C03659=1179.492,110.522,-52.209,-178.814,6.218,148.772
C03660=1179.488,110.772,-52.228,-178.811,6.218,148.772
C03661=1179.483,111.021,-52.246,-178.809,6.220,148.771
C03662=1179.478,111.270,-52.266,-178.806,6.222,148.771
C03663=1179.473,111.519,-52.285,-178.803,6.222,148.770
C03664=1179.468,111.769,-52.304,-178.801,6.224,148.770
C03665=1179.463,112.018,-52.323,-178.799,6.225,148.769
C03666=1179.459,112.267,-52.342,-178.795,6.226,148.769
C03667=1179.453,112.517,-52.361,-178.793,6.228,148.768
C03668=1179.449,112.765,-52.379,-178.790,6.229,148.768
C03669=1179.444,113.015,-52.399,-178.787,6.230,148.767
C03670=1179.439,113.263,-52.418,-178.785,6.232,148.767
C03671=1179.434,113.514,-52.437,-178.782,6.233,148.767
C03672=1179.429,113.762,-52.456,-178.779,6.234,148.766
C03673=1179.425,114.012,-52.475,-178.777,6.236,148.765
C03674=1179.420,114.260,-52.494,-178.774,6.237,148.765
C03675=1179.415,114.510,-52.514,-178.771,6.239,148.764
C03676=1179.410,114.759,-52.532,-178.769,6.240,148.764
C03677=1179.405,115.009,-52.552,-178.766,6.241,148.764
C03678=1179.401,115.257,-52.570,-178.764,6.243,148.763
C03679=1179.396,115.507,-52.590,-178.761,6.244,148.763
C03680=1179.390,115.756,-52.609,-178.758,6.245,148.762
C03681=1179.386,116.005,-52.628,-178.756,6.247,148.762
C03682=1179.382,116.255,-52.648,-178.752,6.248,148.761
C03683=1179.376,116.504,-52.666,-178.750,6.249,148.761
C03684=1179.372,116.753,-52.686,-178.748,6.251,148.760
C03685=1179.367,117.002,-52.705,-178.744,6.252,148.760
C03686=1179.362,117.252,-52.724,-178.742,6.253,148.759
C03687=1179.357,117.501,-52.744,-178.740,6.255,148.759
C03688=1179.353,117.750,-52.763,-178.737,6.257,148.759
C03689=1179.347,117.999,-52.782,-178.734,6.257,148.758
C03690=1179.343,118.248,-52.802,-178.732,6.259,148.757
C03691=1179.339,118.498,-52.821,-178.729,6.261,148.757
C03692=1179.333,118.746,-52.840,-178.726,6.261,148.756
C03693=1179.328,118.996,-52.860,-178.724,6.263,148.756
C03694=1179.323,119.245,-52.879,-178.721,6.265,148.756
C03695=1179.319,119.494,-52.898,-178.718,6.267,148.755
C03696=1179.314,119.744,-52.918,-178.716,6.267,148.755
C03697=1179.309,119.993,-52.937,-178.713,6.269,148.754
C03698=1179.304,120.242,-52.957,-178.710,6.271,148.754
C03699=1179.299,120.491,-52.976,-178.708,6.271,148.753
C03700=1179.295,120.740,-52.995,-178.705,6.273,148.753
C03701=1179.290,120.990,-53.015,-178.702,6.275,148.752
C03702=1179.285,121.239,-53.034,-178.700,6.276,148.752
C03703=1179.280,121.488,-53.054,-178.697,6.277,148.751
C03704=1179.276,121.737,-53.074,-178.694,6.279,148.751
C03705=1179.271,121.986,-53.093,-178.691,6.280,148.751
C03706=1179.266,122.235,-53.112,-178.689,6.281,148.750
C03707=1179.261,122.484,-53.132,-178.686,6.283,148.750
C03708=1179.256,122.734,-53.151,-178.683,6.284,148.749
C03709=1179.251,122.983,-53.171,-178.681,6.285,148.749
C03710=1179.246,123.232,-53.190,-178.679,6.287,148.748
C03711=1179.242,123.481,-53.211,-178.675,6.289,148.748
C03712=1179.238,123.730,-53.230,-178.673,6.290,148.747
C03713=1179.232,123.979,-53.249,-178.671,6.291,148.747
C03714=1179.228,124.229,-53.269,-178.667,6.293,148.746
C03715=1179.223,124.478,-53.288,-178.665,6.294,148.746
C03716=1179.218,124.727,-53.309,-178.663,6.295,148.745
C03717=1179.213,124.976,-53.328,-178.660,6.297,148.745
C03718=1179.208,125.226,-53.348,-178.657,6.298,148.744
C03719=1179.204,125.475,-53.367,-178.654,6.300,148.744
C03720=1179.199,125.724,-53.387,-178.652,6.301,148.744
C03721=1179.194,125.973,-53.407,-178.649,6.303,148.743
C03722=1179.189,126.223,-53.427,-178.646,6.304,148.743
C03723=1179.185,126.472,-53.447,-178.643,6.306,148.742
C03724=1179.179,126.721,-53.466,-178.641,6.307,148.742
C03725=1179.175,126.970,-53.485,-178.638,6.309,148.741
C03726=1179.171,127.219,-53.506,-178.636,6.310,148.741
C03727=1179.165,127.468,-53.525,-178.633,6.312,148.740
C03728=1179.161,127.717,-53.545,-178.630,6.313,148.740
C03729=1179.156,127.966,-53.565,-178.628,6.314,148.740
C03730=1179.152,128.216,-53.585,-178.625,6.316,148.739
C03731=1179.147,128.465,-53.604,-178.622,6.318,148.739
C03732=1179.142,128.714,-53.624,-178.620,6.318,148.738
C03733=1179.137,128.963,-53.644,-178.617,6.320,148.738
C03734=1179.133,129.212,-53.664,-178.614,6.322,148.737
C03735=1179.127,129.462,-53.685,-178.611,6.323,148.737
C03736=1179.122,129.711,-53.704,-178.609,6.324,148.736
C03737=1179.117,129.960,-53.724,-178.606,6.326,148.736
C03738=1179.113,130.209,-53.744,-178.604,6.328,148.736
C03739=1179.108,130.458,-53.764,-178.601,6.329,148.735
C03740=1179.103,130.708,-53.784,-178.598,6.331,148.735
C03741=1179.098,130.956,-53.804,-178.596,6.332,148.734
C03742=1179.094,131.206,-53.824,-178.593,6.334,148.734
C03743=1179.089,131.455,-53.844,-178.590,6.335,148.733
C03744=1179.084,131.704,-53.864,-178.587,6.337,148.733
C03745=1179.080,131.953,-53.884,-178.585,6.338,148.732
C03746=1179.074,132.222,-53.906,-178.582,6.339,148.732
C03747=1179.070,132.490,-53.928,-178.579,6.341,148.732
C03748=1179.064,132.759,-53.949,-178.576,6.343,148.731
C03749=1179.059,133.028,-53.970,-178.574,6.344,148.731
C03750=1179.054,133.277,-53.991,-178.571,6.346,148.730
C03751=1179.049,133.525,-54.011,-178.568,6.347,148.730
C03752=1179.044,133.775,-54.031,-178.565,6.349,148.729
C03753=1179.040,134.024,-54.051,-178.562,6.351,148.729
C03754=1179.035,134.273,-54.071,-178.560,6.352,148.728
C03755=1179.031,134.522,-54.091,-178.558,6.354,148.728
C03756=1179.025,134.772,-54.112,-178.554,6.355,148.727
C03757=1179.021,135.021,-54.132,-178.552,6.357,148.727
C03758=1179.016,135.269,-54.152,-178.549,6.358,148.727
C03759=1179.011,135.518,-54.172,-178.547,6.359,148.726
C03760=1179.006,135.768,-54.192,-178.544,6.361,148.726
C03761=1179.001,136.017,-54.213,-178.541,6.363,148.725
C03762=1178.997,136.266,-54.233,-178.538,6.364,148.725
C03763=1178.992,136.515,-54.254,-178.536,6.366,148.724
C03764=1178.988,136.765,-54.273,-178.533,6.367,148.724
C03765=1178.983,137.014,-54.294,-178.531,6.369,148.724
C03766=1178.978,137.263,-54.315,-178.528,6.370,148.723
C03767=1178.974,137.512,-54.335,-178.525,6.372,148.723
C03768=1178.968,137.762,-54.355,-178.522,6.374,148.722
C03769=1178.964,138.011,-54.376,-178.520,6.375,148.722
C03770=1178.959,138.259,-54.396,-178.517,6.376,148.721
C03771=1178.954,138.508,-54.416,-178.515,6.378,148.721
C03772=1178.949,138.757,-54.437,-178.512,6.380,148.721
C03773=1178.944,139.007,-54.457,-178.509,6.381,148.720
C03774=1178.940,139.256,-54.477,-178.506,6.383,148.720
C03775=1178.935,139.505,-54.498,-178.504,6.384,148.719
C03776=1178.930,139.754,-54.518,-178.501,6.386,148.719
C03777=1178.926,140.003,-54.539,-178.499,6.387,148.719
C03778=1178.921,140.252,-54.560,-178.496,6.389,148.718
C03779=1178.916,140.501,-54.580,-178.493,6.391,148.718
C03780=1178.912,140.750,-54.601,-178.490,6.392,148.717
C03781=1178.906,141.000,-54.621,-178.488,6.393,148.717
C03782=1178.902,141.249,-54.641,-178.485,6.395,148.716
C03783=1178.897,141.498,-54.662,-178.482,6.397,148.716
C03784=1178.892,141.747,-54.682,-178.480,6.398,148.716
C03785=1178.888,141.996,-54.703,-178.477,6.400,148.715
C03786=1178.883,142.245,-54.724,-178.474,6.402,148.715
C03787=1178.878,142.494,-54.744,-178.472,6.403,148.714
C03788=1178.873,142.743,-54.765,-178.469,6.404,148.714
C03789=1178.869,142.992,-54.786,-178.466,6.406,148.713
C03790=1178.864,143.241,-54.806,-178.464,6.408,148.713
C03791=1178.859,143.491,-54.827,-178.461,6.410,148.713
C03792=1178.855,143.739,-54.847,-178.458,6.411,148.712
C03793=1178.849,143.989,-54.868,-178.456,6.413,148.712
C03794=1178.845,144.238,-54.889,-178.453,6.414,148.711
C03795=1178.840,144.488,-54.910,-178.450,6.415,148.711
C03796=1178.836,144.736,-54.931,-178.448,6.417,148.711
C03797=1178.831,144.985,-54.952,-178.445,6.419,148.710
C03798=1178.827,145.234,-54.972,-178.442,6.421,148.710
C03799=1178.821,145.483,-54.993,-178.440,6.422,148.709
C03800=1178.817,145.732,-55.014,-178.437,6.424,148.709
C03801=1178.812,145.982,-55.035,-178.434,6.426,148.709
C03802=1178.807,146.231,-55.055,-178.432,6.427,148.708
C03803=1178.802,146.480,-55.076,-178.429,6.428,148.708
C03804=1178.798,146.728,-55.097,-178.426,6.430,148.707
C03805=1178.793,146.977,-55.118,-178.424,6.432,148.707
C03806=1178.788,147.226,-55.138,-178.421,6.434,148.706
C03807=1178.784,147.476,-55.160,-178.418,6.435,148.706
C03808=1178.779,147.726,-55.181,-178.415,6.437,148.706
C03809=1178.774,147.975,-55.201,-178.413,6.439,148.705
C03810=1178.769,148.223,-55.223,-178.410,6.441,148.705
C03811=1178.765,148.472,-55.243,-178.407,6.441,148.704
C03812=1178.760,148.721,-55.264,-178.405,6.443,148.704
C03813=1178.755,148.971,-55.285,-178.402,6.445,148.704
C03814=1178.751,149.219,-55.306,-178.399,6.446,148.703
C03815=1178.746,149.469,-55.327,-178.397,6.448,148.703
C03816=1178.742,149.718,-55.348,-178.394,6.450,148.702
C03817=1178.737,149.967,-55.370,-178.391,6.452,148.702
C03818=1178.731,150.216,-55.390,-178.389,6.453,148.702
C03819=1178.727,150.465,-55.411,-178.386,6.455,148.701
C03820=1178.722,150.713,-55.433,-178.383,6.457,148.701
C03821=1178.718,150.963,-55.454,-178.381,6.458,148.700
C03822=1178.713,151.212,-55.474,-178.378,6.459,148.700
C03823=1178.708,151.461,-55.496,-178.375,6.461,148.700
C03824=1178.703,151.710,-55.517,-178.373,6.463,148.699
C03825=1178.699,151.959,-55.537,-178.370,6.465,148.699
C03826=1178.694,152.209,-55.559,-178.367,6.466,148.698
C03827=1178.689,152.458,-55.580,-178.365,6.468,148.698
C03828=1178.684,152.706,-55.602,-178.362,6.470,148.698
C03829=1178.680,152.955,-55.622,-178.359,6.472,148.697
C03830=1178.675,153.204,-55.644,-178.356,6.473,148.697
C03831=1178.670,153.454,-55.665,-178.354,6.475,148.696
C03832=1178.665,153.703,-55.686,-178.351,6.477,148.696
C03833=1178.661,153.952,-55.707,-178.349,6.478,148.696
C03834=1178.656,154.201,-55.728,-178.346,6.480,148.695
C03835=1178.652,154.450,-55.750,-178.343,6.481,148.695
C03836=1178.647,154.699,-55.771,-178.340,6.483,148.694
C03837=1178.642,154.948,-55.792,-178.338,6.485,148.694
C03838=1178.637,155.197,-55.813,-178.335,6.486,148.694
C03839=1178.633,155.446,-55.835,-178.332,6.488,148.693
C03840=1178.628,155.695,-55.857,-178.330,6.490,148.693
C03841=1178.623,155.944,-55.878,-178.327,6.492,148.692
C03842=1178.618,156.193,-55.900,-178.324,6.493,148.692
C03843=1178.614,156.443,-55.921,-178.322,6.495,148.692
C03844=1178.609,156.691,-55.942,-178.319,6.497,148.691
C03845=1178.604,156.940,-55.963,-178.316,6.499,148.691
C03846=1178.599,157.189,-55.985,-178.314,6.500,148.691
C03847=1178.595,157.438,-56.007,-178.311,6.502,148.690
C03848=1178.590,157.688,-56.028,-178.308,6.504,148.690
C03849=1178.586,157.936,-56.049,-178.305,6.506,148.689
C03850=1178.580,158.205,-56.072,-178.303,6.507,148.689
C03851=1178.576,158.474,-56.096,-178.300,6.509,148.689
C03852=1178.570,158.743,-56.119,-178.297,6.511,148.688
C03853=1178.566,159.012,-56.142,-178.294,6.512,148.688
C03854=1178.561,159.261,-56.164,-178.292,6.514,148.687
C03855=1178.556,159.510,-56.186,-178.289,6.516,148.687
C03856=1178.551,159.759,-56.207,-178.286,6.518,148.687
C03857=1178.546,160.008,-56.228,-178.284,6.519,148.686
C03858=1178.542,160.257,-56.250,-178.281,6.521,148.686
C03859=1178.537,160.506,-56.272,-178.278,6.523,148.686
C03860=1178.533,160.756,-56.293,-178.275,6.525,148.685
C03861=1178.528,161.005,-56.315,-178.273,6.527,148.685
C03862=1178.523,161.253,-56.337,-178.270,6.528,148.684
C03863=1178.519,161.503,-56.359,-178.267,6.530,148.684
C03864=1178.514,161.751,-56.380,-178.265,6.532,148.684
C03865=1178.509,162.001,-56.401,-178.262,6.534,148.683
C03866=1178.504,162.250,-56.424,-178.259,6.535,148.683
C03867=1178.499,162.499,-56.445,-178.257,6.537,148.683
C03868=1178.495,162.748,-56.467,-178.254,6.539,148.682
C03869=1178.490,162.997,-56.489,-178.251,6.541,148.682
C03870=1178.485,163.245,-56.511,-178.249,6.542,148.681
C03871=1178.481,163.494,-56.533,-178.246,6.544,148.681
C03872=1178.476,163.744,-56.554,-178.243,6.546,148.681
C03873=1178.472,163.993,-56.576,-178.241,6.548,148.680
C03874=1178.467,164.242,-56.597,-178.238,6.549,148.680
C03875=1178.463,164.491,-56.619,-178.235,6.551,148.680
C03876=1178.458,164.740,-56.641,-178.233,6.553,148.679
C03877=1178.453,164.988,-56.663,-178.230,6.555,148.679
C03878=1178.449,165.238,-56.685,-178.227,6.557,148.678
C03879=1178.443,165.487,-56.707,-178.224,6.558,148.678
C03880=1178.439,165.736,-56.729,-178.222,6.560,148.678
C03881=1178.434,165.985,-56.751,-178.219,6.562,148.677
C03882=1178.430,166.234,-56.773,-178.216,6.564,148.677
C03883=1178.425,166.483,-56.795,-178.214,6.565,148.677
C03884=1178.420,166.732,-56.817,-178.211,6.567,148.676
C03885=1178.416,166.981,-56.838,-178.208,6.569,148.676
C03886=1178.411,167.230,-56.860,-178.206,6.571,148.676
C03887=1178.406,167.479,-56.883,-178.203,6.572,148.675
C03888=1178.402,167.728,-56.905,-178.200,6.574,148.675
C03889=1178.397,167.976,-56.927,-178.198,6.576,148.674
C03890=1178.393,168.226,-56.949,-178.195,6.578,148.674
C03891=1178.388,168.474,-56.971,-178.192,6.580,148.674
C03892=1178.383,168.724,-56.993,-178.190,6.581,148.673
C03893=1178.378,168.973,-57.015,-178.187,6.583,148.673
C03894=1178.374,169.222,-57.037,-178.184,6.585,148.673
C03895=1178.369,169.470,-57.059,-178.182,6.587,148.672
C03896=1178.365,169.719,-57.082,-178.179,6.588,148.672
C03897=1178.359,169.968,-57.104,-178.176,6.591,148.672
C03898=1178.355,170.218,-57.126,-178.173,6.593,148.671
C03899=1178.350,170.466,-57.148,-178.170,6.595,148.671
C03900=1178.346,170.715,-57.170,-178.168,6.596,148.670
C03901=1178.340,170.964,-57.193,-178.165,6.598,148.670
C03902=1178.336,171.213,-57.215,-178.163,6.600,148.670
C03903=1178.331,171.462,-57.236,-178.160,6.602,148.670
C03904=1178.326,171.711,-57.259,-178.157,6.604,148.669
C03905=1178.322,171.960,-57.282,-178.155,6.606,148.669
C03906=1178.318,172.209,-57.303,-178.152,6.607,148.668
C03907=1178.313,172.458,-57.326,-178.149,6.609,148.668
C03908=1178.308,172.706,-57.349,-178.147,6.611,148.668
C03909=1178.304,172.956,-57.371,-178.144,6.613,148.667
C03910=1178.299,173.205,-57.393,-178.141,6.614,148.667
C03911=1178.294,173.453,-57.416,-178.139,6.616,148.667
C03912=1178.290,173.703,-57.438,-178.136,6.618,148.666
C03913=1178.285,173.951,-57.459,-178.133,6.620,148.666
C03914=1178.280,174.201,-57.483,-178.131,6.621,148.666
C03915=1178.276,174.450,-57.505,-178.127,6.624,148.665
C03916=1178.270,174.699,-57.527,-178.125,6.626,148.665
C03917=1178.266,174.948,-57.550,-178.122,6.628,148.665
C03918=1178.262,175.197,-57.572,-178.120,6.630,148.664
C03919=1178.257,175.445,-57.595,-178.117,6.631,148.664
C03920=1178.253,175.695,-57.617,-178.114,6.633,148.664
C03921=1178.247,175.943,-57.640,-178.112,6.635,148.663
C03922=1178.243,176.192,-57.662,-178.109,6.637,148.663
C03923=1178.239,176.442,-57.684,-178.106,6.639,148.663
C03924=1178.233,176.690,-57.707,-178.104,6.640,148.662
C03925=1178.229,176.939,-57.729,-178.101,6.642,148.662
C03926=1178.224,177.188,-57.752,-178.098,6.644,148.661
C03927=1178.220,177.436,-57.775,-178.095,6.647,148.661
C03928=1178.215,177.686,-57.797,-178.093,6.649,148.661
C03929=1178.211,177.935,-57.820,-178.090,6.650,148.661
C03930=1178.206,178.184,-57.843,-178.087,6.652,148.660
C03931=1178.201,178.432,-57.865,-178.085,6.654,148.660
C03932=1178.196,178.682,-57.888,-178.082,6.656,148.659
C03933=1178.192,178.931,-57.911,-178.079,6.658,148.659
C03934=1178.187,179.180,-57.933,-178.077,6.659,148.659
C03935=1178.183,179.428,-57.956,-178.074,6.661,148.658
C03936=1178.178,179.677,-57.979,-178.071,6.663,148.658
C03937=1178.174,179.927,-58.001,-178.069,6.666,148.658
C03938=1178.169,180.175,-58.024,-178.066,6.668,148.658
C03939=1178.165,180.424,-58.047,-178.063,6.669,148.657
C03940=1178.160,180.673,-58.069,-178.061,6.671,148.657
C03941=1178.156,180.922,-58.092,-178.058,6.673,148.656
C03942=1178.150,181.170,-58.115,-178.055,6.675,148.656
C03943=1178.145,181.420,-58.138,-178.053,6.676,148.656
C03944=1178.141,181.669,-58.161,-178.050,6.678,148.655
C03945=1178.137,181.918,-58.184,-178.047,6.681,148.655
C03946=1178.132,182.166,-58.206,-178.044,6.683,148.655
C03947=1178.127,182.416,-58.229,-178.042,6.685,148.655
C03948=1178.122,182.665,-58.252,-178.039,6.686,148.654
C03949=1178.118,182.913,-58.275,-178.036,6.688,148.654
C03950=1178.113,183.162,-58.298,-178.034,6.690,148.654
C03951=1178.109,183.411,-58.320,-178.031,6.692,148.653
C03952=1178.104,183.660,-58.344,-178.029,6.694,148.653
C03953=1178.099,183.909,-58.367,-178.026,6.697,148.653
C03954=1178.095,184.179,-58.391,-178.023,6.698,148.652
C03955=1178.090,184.448,-58.416,-178.020,6.700,148.652
C03956=1178.084,184.718,-58.441,-178.017,6.703,148.652
C03957=1178.080,184.987,-58.467,-178.014,6.704,148.651
C03958=1178.075,185.237,-58.489,-178.012,6.706,148.651
C03959=1178.070,185.486,-58.513,-178.008,6.709,148.651
C03960=1178.066,185.734,-58.535,-178.006,6.711,148.650
C03961=1178.061,185.983,-58.558,-178.003,6.712,148.650
C03962=1178.056,186.232,-58.582,-178.000,6.714,148.650
C03963=1178.052,186.481,-58.605,-177.998,6.716,148.649
C03964=1178.048,186.729,-58.628,-177.996,6.718,148.649
C03965=1178.043,186.978,-58.651,-177.993,6.720,148.649
C03966=1178.038,187.227,-58.675,-177.990,6.722,148.648
C03967=1178.033,187.476,-58.698,-177.987,6.724,148.648
C03968=1178.029,187.725,-58.720,-177.984,6.726,148.648
C03969=1178.024,187.974,-58.744,-177.982,6.728,148.648
C03970=1178.020,188.223,-58.767,-177.979,6.730,148.647
C03971=1178.015,188.472,-58.790,-177.977,6.732,148.647
C03972=1178.010,188.721,-58.814,-177.974,6.734,148.646
C03973=1178.006,188.969,-58.836,-177.971,6.736,148.646
C03974=1178.002,189.218,-58.860,-177.969,6.738,148.646
C03975=1177.997,189.467,-58.883,-177.966,6.740,148.646
C03976=1177.992,189.716,-58.907,-177.963,6.742,148.645
C03977=1177.987,189.965,-58.930,-177.960,6.744,148.645
C03978=1177.982,190.214,-58.953,-177.957,6.746,148.645
C03979=1177.978,190.463,-58.976,-177.955,6.748,148.644
C03980=1177.974,190.711,-59.000,-177.953,6.750,148.644
C03981=1177.969,190.960,-59.023,-177.950,6.752,148.644
C03982=1177.964,191.209,-59.046,-177.947,6.754,148.643
C03983=1177.960,191.458,-59.070,-177.944,6.756,148.643
C03984=1177.955,191.707,-59.093,-177.942,6.758,148.643
C03985=1177.950,191.956,-59.117,-177.939,6.760,148.643
C03986=1177.946,192.205,-59.141,-177.936,6.762,148.642
C03987=1177.941,192.454,-59.164,-177.934,6.764,148.642
C03988=1177.936,192.703,-59.187,-177.930,6.766,148.642
C03989=1177.932,192.952,-59.211,-177.928,6.768,148.641
C03990=1177.927,193.200,-59.235,-177.926,6.770,148.641
C03991=1177.923,193.449,-59.258,-177.923,6.772,148.641
C03992=1177.919,193.698,-59.281,-177.920,6.774,148.640
C03993=1177.914,193.947,-59.304,-177.917,6.776,148.640
C03994=1177.910,194.195,-59.328,-177.915,6.779,148.640
C03995=1177.905,194.444,-59.352,-177.912,6.780,148.640
C03996=1177.900,194.693,-59.375,-177.910,6.782,148.639
C03997=1177.896,194.942,-59.399,-177.906,6.785,148.639
C03998=1177.891,195.191,-59.422,-177.904,6.787,148.639
C03999=1177.886,195.440,-59.446,-177.901,6.789,148.638
C04000=1177.882,195.688,-59.470,-177.899,6.790,148.638
C04001=1177.877,195.937,-59.493,-177.896,6.792,148.638
C04002=1177.873,196.186,-59.517,-177.893,6.795,148.638
C04003=1177.868,196.435,-59.541,-177.891,6.797,148.637
C04004=1177.863,196.684,-59.565,-177.888,6.799,148.637
C04005=1177.858,196.932,-59.589,-177.885,6.801,148.637
C04006=1177.854,197.181,-59.612,-177.883,6.803,148.636
C04007=1177.849,197.431,-59.635,-177.880,6.805,148.636
C04008=1177.845,197.679,-59.660,-177.877,6.807,148.636
C04009=1177.840,197.928,-59.683,-177.875,6.809,148.635
C04010=1177.836,198.176,-59.707,-177.872,6.812,148.635
C04011=1177.831,198.426,-59.731,-177.869,6.814,148.635
C04012=1177.827,198.675,-59.755,-177.866,6.815,148.635
C04013=1177.822,198.924,-59.778,-177.864,6.817,148.634
C04014=1177.817,199.172,-59.803,-177.862,6.819,148.634
C04015=1177.813,199.421,-59.826,-177.858,6.822,148.634
C04016=1177.808,199.670,-59.850,-177.856,6.824,148.633
C04017=1177.804,199.918,-59.874,-177.853,6.825,148.633
C04018=1177.799,200.167,-59.898,-177.851,6.828,148.633
C04019=1177.795,200.416,-59.922,-177.848,6.830,148.633
C04020=1177.791,200.665,-59.945,-177.845,6.832,148.632
C04021=1177.785,200.914,-59.970,-177.842,6.834,148.632
C04022=1177.781,201.162,-59.994,-177.839,6.837,148.632
C04023=1177.776,201.411,-60.018,-177.837,6.839,148.632
C04024=1177.772,201.660,-60.042,-177.834,6.840,148.631
C04025=1177.767,201.909,-60.065,-177.832,6.842,148.631
C04026=1177.762,202.158,-60.090,-177.829,6.845,148.631
C04027=1177.758,202.407,-60.114,-177.826,6.847,148.630
C04028=1177.754,202.656,-60.137,-177.823,6.849,148.630
C04029=1177.749,202.904,-60.162,-177.821,6.851,148.630
C04030=1177.744,203.153,-60.186,-177.818,6.853,148.630
C04031=1177.740,203.401,-60.210,-177.815,6.855,148.629
C04032=1177.736,203.651,-60.234,-177.813,6.857,148.629
C04033=1177.731,203.899,-60.258,-177.810,6.859,148.629
C04034=1177.726,204.148,-60.283,-177.807,6.862,148.628
C04035=1177.722,204.397,-60.307,-177.805,6.864,148.628
C04036=1177.717,204.646,-60.330,-177.802,6.866,148.628
C04037=1177.712,204.895,-60.355,-177.799,6.868,148.628
C04038=1177.708,205.143,-60.379,-177.796,6.870,148.627
C04039=1177.704,205.392,-60.403,-177.794,6.872,148.627
C04040=1177.699,205.641,-60.428,-177.792,6.874,148.627
C04041=1177.694,205.889,-60.452,-177.788,6.877,148.627
C04042=1177.690,206.139,-60.476,-177.786,6.879,148.626
C04043=1177.685,206.387,-60.501,-177.784,6.880,148.626
C04044=1177.680,206.636,-60.525,-177.780,6.883,148.626
C04045=1177.676,206.884,-60.549,-177.778,6.885,148.626
C04046=1177.672,207.134,-60.574,-177.775,6.887,148.625
C04047=1177.667,207.382,-60.598,-177.772,6.890,148.625
C04048=1177.662,207.631,-60.622,-177.770,6.892,148.625
C04049=1177.658,207.879,-60.647,-177.767,6.894,148.625
C04050=1177.654,208.128,-60.671,-177.764,6.896,148.624
C04051=1177.649,208.377,-60.696,-177.762,6.898,148.624
C04052=1177.644,208.626,-60.720,-177.759,6.900,148.624
C04053=1177.640,208.875,-60.745,-177.757,6.902,148.623
C04054=1177.635,209.123,-60.769,-177.754,6.905,148.623
C04055=1177.630,209.372,-60.793,-177.751,6.907,148.623
C04056=1177.626,209.620,-60.818,-177.749,6.908,148.623
C04057=1177.621,209.870,-60.843,-177.746,6.911,148.623
C04058=1177.616,210.141,-60.869,-177.743,6.913,148.622
C04059=1177.611,210.411,-60.895,-177.740,6.916,148.622
C04060=1177.607,210.681,-60.922,-177.737,6.918,148.622
C04061=1177.602,210.952,-60.948,-177.734,6.920,148.621
C04062=1177.597,211.200,-60.973,-177.731,6.923,148.621
C04063=1177.593,211.449,-60.998,-177.729,6.925,148.621
C04064=1177.588,211.698,-61.022,-177.726,6.927,148.621
C04065=1177.583,211.947,-61.046,-177.723,6.930,148.620
C04066=1177.579,212.195,-61.072,-177.720,6.931,148.620
C04067=1177.575,212.444,-61.096,-177.718,6.934,148.620
C04068=1177.570,212.693,-61.121,-177.715,6.936,148.620
C04069=1177.565,212.942,-61.146,-177.712,6.938,148.619
C04070=1177.561,213.190,-61.170,-177.710,6.940,148.619
C04071=1177.556,213.440,-61.195,-177.707,6.943,148.619
C04072=1177.552,213.688,-61.220,-177.705,6.945,148.619
C04073=1177.547,213.936,-61.244,-177.702,6.947,148.618
C04074=1177.542,214.186,-61.269,-177.699,6.949,148.618
C04075=1177.538,214.434,-61.294,-177.697,6.951,148.618
C04076=1177.534,214.683,-61.319,-177.694,6.953,148.618
C04077=1177.529,214.931,-61.343,-177.691,6.956,148.617
C04078=1177.524,215.180,-61.368,-177.689,6.958,148.617
C04079=1177.520,215.430,-61.393,-177.686,6.960,148.617
C04080=1177.516,215.677,-61.418,-177.683,6.963,148.617
C04081=1177.511,215.927,-61.443,-177.681,6.965,148.616
C04082=1177.506,216.175,-61.468,-177.677,6.967,148.616
C04083=1177.502,216.424,-61.493,-177.675,6.969,148.616
C04084=1177.497,216.673,-61.517,-177.672,6.971,148.616
C04085=1177.492,216.921,-61.543,-177.670,6.974,148.616
C04086=1177.489,217.170,-61.567,-177.667,6.976,148.615
C04087=1177.484,217.419,-61.592,-177.664,6.978,148.615
C04088=1177.479,217.667,-61.618,-177.662,6.981,148.615
C04089=1177.474,217.916,-61.642,-177.659,6.982,148.615
C04090=1177.471,218.165,-61.667,-177.657,6.985,148.614
C04091=1177.466,218.413,-61.692,-177.654,6.987,148.614
C04092=1177.461,218.663,-61.717,-177.651,6.989,148.614
C04093=1177.456,218.911,-61.743,-177.648,6.992,148.614
C04094=1177.452,219.160,-61.767,-177.645,6.994,148.613
C04095=1177.448,219.408,-61.792,-177.643,6.996,148.613
C04096=1177.443,219.658,-61.817,-177.640,6.998,148.613
C04097=1177.438,219.906,-61.843,-177.638,7.001,148.613
C04098=1177.434,220.155,-61.867,-177.635,7.003,148.613
C04099=1177.430,220.403,-61.893,-177.632,7.005,148.612
C04100=1177.425,220.652,-61.918,-177.630,7.007,148.612
C04101=1177.420,220.900,-61.943,-177.627,7.010,148.612
C04102=1177.416,221.149,-61.969,-177.624,7.012,148.612
C04103=1177.412,221.398,-61.993,-177.621,7.015,148.611
C04104=1177.407,221.646,-62.019,-177.619,7.017,148.611
C04105=1177.403,221.896,-62.044,-177.616,7.019,148.611
C04106=1177.398,222.144,-62.069,-177.613,7.021,148.611
C04107=1177.394,222.393,-62.095,-177.611,7.023,148.610
C04108=1177.389,222.641,-62.119,-177.608,7.026,148.610
C04109=1177.384,222.890,-62.145,-177.606,7.028,148.610
C04110=1177.380,223.138,-62.171,-177.603,7.030,148.610
C04111=1177.376,223.387,-62.195,-177.600,7.033,148.610
C04112=1177.372,223.636,-62.221,-177.597,7.035,148.609
C04113=1177.367,223.884,-62.246,-177.595,7.038,148.609
C04114=1177.362,224.134,-62.271,-177.592,7.039,148.609
C04115=1177.357,224.382,-62.297,-177.589,7.042,148.609
C04116=1177.353,224.631,-62.322,-177.587,7.044,148.609
C04117=1177.349,224.880,-62.348,-177.584,7.046,148.608
C04118=1177.344,225.128,-62.373,-177.581,7.049,148.608
C04119=1177.340,225.377,-62.399,-177.579,7.051,148.608
C04120=1177.335,225.625,-62.424,-177.576,7.054,148.608
C04121=1177.331,225.874,-62.450,-177.574,7.056,148.608
C04122=1177.326,226.123,-62.475,-177.570,7.058,148.607
C04123=1177.321,226.371,-62.500,-177.568,7.060,148.607
C04124=1177.317,226.620,-62.526,-177.566,7.062,148.607
C04125=1177.313,226.869,-62.552,-177.562,7.065,148.607
C04126=1177.308,227.117,-62.577,-177.560,7.067,148.606
C04127=1177.304,227.366,-62.603,-177.557,7.070,148.606
C04128=1177.300,227.615,-62.628,-177.555,7.072,148.606
C04129=1177.295,227.863,-62.654,-177.552,7.074,148.606
C04130=1177.290,228.112,-62.680,-177.549,7.077,148.606
C04131=1177.286,228.361,-62.705,-177.546,7.079,148.605
C04132=1177.281,228.609,-62.730,-177.544,7.081,148.605
C04133=1177.277,228.858,-62.756,-177.542,7.084,148.605
C04134=1177.273,229.107,-62.782,-177.539,7.086,148.605
C04135=1177.268,229.355,-62.807,-177.536,7.088,148.605
C04136=1177.263,229.604,-62.833,-177.533,7.091,148.604
C04137=1177.259,229.853,-62.859,-177.531,7.093,148.604
C04138=1177.254,230.102,-62.885,-177.528,7.096,148.604
C04139=1177.250,230.350,-62.910,-177.526,7.098,148.604
C04140=1177.245,230.599,-62.936,-177.522,7.100,148.604
C04141=1177.241,230.847,-62.962,-177.520,7.103,148.603
C04142=1177.237,231.095,-62.988,-177.517,7.105,148.603
C04143=1177.232,231.344,-63.014,-177.515,7.107,148.603
C04144=1177.227,231.593,-63.040,-177.512,7.110,148.603
C04145=1177.223,231.842,-63.066,-177.509,7.112,148.603
C04146=1177.218,232.090,-63.091,-177.507,7.114,148.602
C04147=1177.214,232.339,-63.117,-177.504,7.117,148.602
C04148=1177.210,232.587,-63.142,-177.502,7.119,148.602
C04149=1177.205,232.836,-63.169,-177.499,7.122,148.602
C04150=1177.200,233.085,-63.194,-177.496,7.124,148.602
C04151=1177.196,233.333,-63.221,-177.493,7.126,148.601
C04152=1177.192,233.582,-63.246,-177.491,7.129,148.601
C04153=1177.187,233.831,-63.273,-177.488,7.131,148.601
C04154=1177.183,234.079,-63.299,-177.486,7.133,148.601
C04155=1177.178,234.328,-63.324,-177.482,7.136,148.601
C04156=1177.174,234.576,-63.350,-177.480,7.138,148.601
C04157=1177.169,234.825,-63.377,-177.477,7.141,148.600
C04158=1177.165,235.074,-63.402,-177.475,7.143,148.600
C04159=1177.161,235.322,-63.428,-177.472,7.146,148.600
C04160=1177.156,235.570,-63.454,-177.469,7.148,148.600
C04161=1177.151,235.819,-63.481,-177.467,7.151,148.600
C04162=1177.147,236.091,-63.509,-177.463,7.153,148.599
C04163=1177.142,236.362,-63.537,-177.461,7.156,148.599
C04164=1177.137,236.634,-63.566,-177.458,7.158,148.599
C04165=1177.132,236.906,-63.595,-177.455,7.161,148.599
C04166=1177.128,237.155,-63.621,-177.452,7.164,148.599
C04167=1177.123,237.402,-63.647,-177.450,7.166,148.599
C04168=1177.119,237.651,-63.673,-177.447,7.169,148.598
C04169=1177.114,237.900,-63.699,-177.444,7.171,148.598
C04170=1177.110,238.148,-63.726,-177.442,7.174,148.598
C04171=1177.105,238.397,-63.752,-177.439,7.175,148.598
C04172=1177.101,238.646,-63.779,-177.436,7.178,148.598
C04173=1177.097,238.895,-63.804,-177.434,7.180,148.598
C04174=1177.093,239.143,-63.831,-177.431,7.183,148.597
C04175=1177.087,239.391,-63.857,-177.429,7.185,148.597
C04176=1177.083,239.639,-63.883,-177.426,7.188,148.597
C04177=1177.078,239.888,-63.910,-177.423,7.190,148.597
C04178=1177.074,240.137,-63.936,-177.421,7.193,148.597
C04179=1177.069,240.386,-63.962,-177.417,7.196,148.596
C04180=1177.065,240.634,-63.989,-177.415,7.198,148.596
C04181=1177.060,240.883,-64.015,-177.412,7.201,148.596
C04182=1177.057,241.131,-64.042,-177.410,7.203,148.596
C04183=1177.052,241.380,-64.068,-177.407,7.205,148.596
C04184=1177.048,241.629,-64.095,-177.405,7.208,148.596
C04185=1177.043,241.878,-64.121,-177.402,7.210,148.596
C04186=1177.039,242.126,-64.147,-177.399,7.212,148.595
C04187=1177.034,242.374,-64.174,-177.397,7.215,148.595
C04188=1177.030,242.623,-64.200,-177.394,7.217,148.595
C04189=1177.025,242.872,-64.227,-177.391,7.220,148.595
C04190=1177.021,243.120,-64.254,-177.389,7.223,148.595
C04191=1177.016,243.368,-64.280,-177.386,7.225,148.595
C04192=1177.012,243.616,-64.306,-177.383,7.228,148.595
C04193=1177.007,243.865,-64.333,-177.381,7.230,148.594
C04194=1177.003,244.114,-64.359,-177.378,7.233,148.594
C04195=1176.998,244.362,-64.386,-177.376,7.235,148.594
C04196=1176.994,244.611,-64.413,-177.373,7.238,148.594
C04197=1176.990,244.859,-64.440,-177.370,7.240,148.594
C04198=1176.985,245.109,-64.466,-177.367,7.243,148.594
C04199=1176.981,245.357,-64.493,-177.365,7.246,148.594
C04200=1176.977,245.605,-64.520,-177.362,7.247,148.593
C04201=1176.972,245.854,-64.547,-177.359,7.250,148.593
C04202=1176.968,246.103,-64.573,-177.357,7.252,148.593
C04203=1176.963,246.351,-64.600,-177.354,7.255,148.593
C04204=1176.959,246.600,-64.627,-177.351,7.258,148.593
C04205=1176.955,246.848,-64.653,-177.349,7.260,148.593
C04206=1176.950,247.096,-64.680,-177.346,7.263,148.593
C04207=1176.945,247.345,-64.707,-177.344,7.265,148.592
C04208=1176.941,247.593,-64.734,-177.341,7.268,148.592
C04209=1176.936,247.842,-64.760,-177.338,7.271,148.592
C04210=1176.932,248.091,-64.787,-177.335,7.273,148.592
C04211=1176.928,248.339,-64.814,-177.333,7.276,148.592
C04212=1176.923,248.587,-64.841,-177.331,7.278,148.592
C04213=1176.919,248.836,-64.868,-177.328,7.281,148.592
C04214=1176.914,249.084,-64.895,-177.325,7.283,148.591
C04215=1176.911,249.333,-64.922,-177.322,7.286,148.591
C04216=1176.906,249.582,-64.949,-177.320,7.289,148.591
C04217=1176.901,249.830,-64.976,-177.318,7.291,148.591
C04218=1176.897,250.079,-65.003,-177.314,7.293,148.591
C04219=1176.893,250.327,-65.029,-177.312,7.296,148.591
C04220=1176.888,250.575,-65.056,-177.309,7.298,148.591
C04221=1176.883,250.824,-65.083,-177.307,7.301,148.590
C04222=1176.879,251.072,-65.111,-177.304,7.303,148.590
C04223=1176.874,251.321,-65.138,-177.301,7.306,148.590
C04224=1176.871,251.570,-65.164,-177.298,7.309,148.590
C04225=1176.866,251.818,-65.191,-177.296,7.311,148.590
C04226=1176.861,252.067,-65.219,-177.293,7.314,148.590
C04227=1176.857,252.315,-65.246,-177.291,7.316,148.590
C04228=1176.852,252.563,-65.273,-177.288,7.319,148.590
C04229=1176.848,252.812,-65.300,-177.285,7.322,148.589
C04230=1176.844,253.061,-65.328,-177.283,7.324,148.589
C04231=1176.840,253.309,-65.354,-177.280,7.327,148.589
C04232=1176.835,253.557,-65.381,-177.277,7.330,148.589
C04233=1176.831,253.805,-65.409,-177.275,7.332,148.589
C04234=1176.826,254.054,-65.436,-177.272,7.335,148.589
C04235=1176.822,254.303,-65.464,-177.269,7.338,148.589
C04236=1176.817,254.552,-65.491,-177.267,7.340,148.589
C04237=1176.813,254.800,-65.518,-177.264,7.343,148.588
C04238=1176.808,255.048,-65.546,-177.262,7.345,148.588
C04239=1176.804,255.296,-65.573,-177.259,7.347,148.588
C04240=1176.800,255.546,-65.600,-177.256,7.350,148.588
C04241=1176.795,255.793,-65.628,-177.254,7.353,148.588
C04242=1176.791,256.042,-65.655,-177.251,7.356,148.588
C04243=1176.786,256.290,-65.682,-177.248,7.359,148.588
C04244=1176.782,256.540,-65.709,-177.246,7.361,148.588
C04245=1176.778,256.788,-65.737,-177.243,7.363,148.587
C04246=1176.773,257.036,-65.764,-177.240,7.366,148.587
C04247=1176.769,257.284,-65.792,-177.238,7.368,148.587
C04248=1176.765,257.533,-65.819,-177.235,7.371,148.587
C04249=1176.760,257.782,-65.847,-177.233,7.374,148.587
C04250=1176.756,258.029,-65.874,-177.230,7.376,148.587
C04251=1176.751,258.278,-65.901,-177.227,7.379,148.587
C04252=1176.747,258.527,-65.929,-177.225,7.382,148.587
C04253=1176.743,258.775,-65.957,-177.222,7.384,148.587
C04254=1176.738,259.024,-65.984,-177.220,7.387,148.587
C04255=1176.734,259.272,-66.012,-177.217,7.390,148.587
C04256=1176.729,259.521,-66.039,-177.214,7.392,148.586
C04257=1176.725,259.768,-66.067,-177.212,7.395,148.586
C04258=1176.721,260.018,-66.094,-177.209,7.398,148.586
C04259=1176.717,260.266,-66.122,-177.207,7.400,148.586
C04260=1176.712,260.514,-66.149,-177.204,7.403,148.586
C04261=1176.708,260.763,-66.178,-177.201,7.406,148.586
C04262=1176.703,261.011,-66.205,-177.199,7.408,148.586
C04263=1176.699,261.259,-66.232,-177.196,7.411,148.586
C04264=1176.695,261.508,-66.261,-177.193,7.414,148.586
C04265=1176.690,261.756,-66.288,-177.191,7.416,148.585
C04266=1176.686,262.030,-66.318,-177.188,7.419,148.585
C04267=1176.680,262.302,-66.349,-177.185,7.423,148.585
C04268=1176.676,262.576,-66.379,-177.182,7.425,148.585
C04269=1176.670,262.848,-66.410,-177.179,7.428,148.585
C04270=1176.667,263.097,-66.438,-177.177,7.431,148.585
C04271=1176.662,263.345,-66.466,-177.174,7.434,148.585
C04272=1176.658,263.593,-66.494,-177.171,7.437,148.585
C04273=1176.653,263.842,-66.521,-177.169,7.439,148.585
C04274=1176.649,264.090,-66.549,-177.166,7.442,148.585
C04275=1176.645,264.339,-66.577,-177.163,7.444,148.584
C04276=1176.640,264.587,-66.604,-177.160,7.447,148.584
C04277=1176.636,264.836,-66.633,-177.158,7.449,148.584
C04278=1176.631,265.084,-66.661,-177.155,7.452,148.584
C04279=1176.627,265.332,-66.689,-177.153,7.455,148.584
C04280=1176.622,265.581,-66.717,-177.151,7.458,148.584
C04281=1176.618,265.829,-66.744,-177.148,7.460,148.584
C04282=1176.614,266.078,-66.773,-177.145,7.463,148.584
C04283=1176.610,266.326,-66.800,-177.142,7.466,148.584
C04284=1176.605,266.574,-66.829,-177.140,7.469,148.584
C04285=1176.601,266.822,-66.857,-177.137,7.472,148.584
C04286=1176.597,267.072,-66.884,-177.134,7.474,148.584
C04287=1176.592,267.320,-66.913,-177.132,7.476,148.584
C04288=1176.588,267.568,-66.940,-177.129,7.479,148.583
C04289=1176.583,267.816,-66.969,-177.127,7.482,148.583
C04290=1176.579,268.064,-66.997,-177.124,7.485,148.583
C04291=1176.575,268.313,-67.025,-177.122,7.487,148.583
C04292=1176.570,268.561,-67.053,-177.119,7.490,148.583
C04293=1176.566,268.810,-67.082,-177.116,7.493,148.583
C04294=1176.562,269.058,-67.109,-177.113,7.496,148.583
C04295=1176.557,269.306,-67.138,-177.111,7.499,148.583
C04296=1176.553,269.554,-67.166,-177.108,7.501,148.583
C04297=1176.548,269.803,-67.195,-177.106,7.504,148.583
C04298=1176.544,270.051,-67.222,-177.104,7.507,148.583
C04299=1176.540,270.300,-67.251,-177.101,7.510,148.583
C04300=1176.536,270.549,-67.279,-177.098,7.513,148.583
C04301=1176.531,270.797,-67.308,-177.095,7.516,148.583
C04302=1176.527,271.045,-67.336,-177.093,7.518,148.583
C04303=1176.523,271.293,-67.364,-177.090,7.521,148.583
C04304=1176.518,271.542,-67.392,-177.087,7.523,148.582
C04305=1176.514,271.790,-67.420,-177.085,7.526,148.582
C04306=1176.510,272.038,-67.450,-177.082,7.528,148.582
C04307=1176.505,272.286,-67.477,-177.080,7.531,148.582
C04308=1176.501,272.535,-67.506,-177.077,7.534,148.582
C04309=1176.496,272.784,-67.535,-177.074,7.537,148.582
C04310=1176.492,273.032,-67.563,-177.072,7.540,148.582
C04311=1176.487,273.281,-67.591,-177.069,7.543,148.582
C04312=1176.483,273.528,-67.620,-177.066,7.545,148.582
C04313=1176.479,273.777,-67.649,-177.064,7.548,148.582
C04314=1176.475,274.025,-67.676,-177.061,7.551,148.582
C04315=1176.470,274.274,-67.705,-177.059,7.554,148.582
C04316=1176.466,274.522,-67.733,-177.056,7.557,148.582
C04317=1176.462,274.770,-67.762,-177.053,7.560,148.582
C04318=1176.457,275.019,-67.791,-177.051,7.563,148.582
C04319=1176.453,275.267,-67.819,-177.048,7.565,148.582
C04320=1176.449,275.515,-67.848,-177.046,7.568,148.581
C04321=1176.445,275.763,-67.876,-177.043,7.571,148.581
C04322=1176.440,276.012,-67.905,-177.040,7.574,148.581
C04323=1176.436,276.260,-67.934,-177.038,7.577,148.581
C04324=1176.432,276.508,-67.962,-177.035,7.579,148.581
C04325=1176.427,276.757,-67.991,-177.033,7.582,148.581
C04326=1176.423,277.005,-68.020,-177.030,7.585,148.581
C04327=1176.419,277.253,-68.048,-177.027,7.588,148.581
C04328=1176.415,277.502,-68.078,-177.025,7.590,148.581
C04329=1176.410,277.750,-68.106,-177.022,7.593,148.581
C04330=1176.406,277.998,-68.134,-177.020,7.596,148.581
C04331=1176.402,278.247,-68.164,-177.017,7.599,148.581
C04332=1176.396,278.495,-68.192,-177.014,7.602,148.581
C04333=1176.392,278.743,-68.222,-177.012,7.604,148.581
C04334=1176.389,278.992,-68.250,-177.010,7.607,148.581
C04335=1176.384,279.239,-68.279,-177.007,7.610,148.581
C04336=1176.379,279.488,-68.308,-177.004,7.613,148.581
C04337=1176.375,279.736,-68.337,-177.001,7.616,148.581
C04338=1176.371,279.985,-68.365,-176.999,7.618,148.581
C04339=1176.367,280.233,-68.394,-176.996,7.621,148.581
C04340=1176.362,280.481,-68.424,-176.994,7.624,148.581
C04341=1176.358,280.730,-68.452,-176.991,7.627,148.581
C04342=1176.354,280.978,-68.481,-176.988,7.630,148.581
C04343=1176.349,281.226,-68.510,-176.986,7.632,148.581
C04344=1176.345,281.474,-68.539,-176.983,7.635,148.581
C04345=1176.341,281.722,-68.569,-176.981,7.638,148.580
C04346=1176.337,281.971,-68.597,-176.978,7.641,148.580
C04347=1176.332,282.219,-68.626,-176.975,7.644,148.580
C04348=1176.327,282.468,-68.655,-176.973,7.646,148.580
C04349=1176.324,282.716,-68.684,-176.971,7.650,148.580
C04350=1176.320,282.964,-68.713,-176.968,7.653,148.580
C04351=1176.315,283.212,-68.743,-176.965,7.656,148.580
C04352=1176.310,283.460,-68.771,-176.963,7.659,148.580
C04353=1176.306,283.709,-68.801,-176.960,7.662,148.580
C04354=1176.302,283.957,-68.830,-176.958,7.664,148.580
C04355=1176.298,284.205,-68.860,-176.955,7.667,148.580
C04356=1176.293,284.453,-68.888,-176.952,7.670,148.580
C04357=1176.289,284.702,-68.917,-176.949,7.673,148.580
C04358=1176.284,284.950,-68.947,-176.947,7.676,148.580
C04359=1176.280,285.198,-68.976,-176.944,7.679,148.580
C04360=1176.276,285.447,-69.004,-176.942,7.681,148.580
C04361=1176.272,285.695,-69.034,-176.940,7.684,148.580
C04362=1176.267,285.943,-69.063,-176.937,7.687,148.580
C04363=1176.263,286.191,-69.092,-176.934,7.690,148.580
C04364=1176.259,286.439,-69.122,-176.931,7.693,148.580
C04365=1176.255,286.687,-69.151,-176.929,7.696,148.580
C04366=1176.251,286.936,-69.181,-176.926,7.698,148.580
C04367=1176.247,287.184,-69.210,-176.924,7.701,148.580
C04368=1176.242,287.432,-69.240,-176.921,7.704,148.580
C04369=1176.238,287.681,-69.268,-176.919,7.708,148.580
C04370=1176.233,287.955,-69.301,-176.916,7.710,148.580
C04371=1176.228,288.231,-69.334,-176.913,7.713,148.580
C04372=1176.223,288.504,-69.366,-176.910,7.717,148.580
C04373=1176.218,288.780,-69.399,-176.907,7.720,148.580
C04374=1176.214,289.028,-69.428,-176.904,7.723,148.580
C04375=1176.210,289.276,-69.458,-176.902,7.726,148.580
C04376=1176.206,289.524,-69.487,-176.899,7.729,148.580
C04377=1176.202,289.773,-69.517,-176.897,7.731,148.580
C04378=1176.197,290.021,-69.546,-176.894,7.734,148.580
C04379=1176.193,290.269,-69.577,-176.892,7.738,148.580
C04380=1176.189,290.517,-69.606,-176.889,7.741,148.580
C04381=1176.184,290.765,-69.636,-176.886,7.744,148.580
C04382=1176.180,291.014,-69.665,-176.884,7.747,148.580
C04383=1176.176,291.262,-69.695,-176.881,7.750,148.580
C04384=1176.171,291.510,-69.724,-176.879,7.752,148.580
C04385=1176.167,291.758,-69.753,-176.876,7.755,148.580
C04386=1176.162,292.006,-69.783,-176.874,7.758,148.580
C04387=1176.158,292.254,-69.814,-176.871,7.761,148.580
C04388=1176.154,292.502,-69.843,-176.868,7.764,148.580
C04389=1176.150,292.751,-69.873,-176.865,7.767,148.580
C04390=1176.146,292.999,-69.902,-176.863,7.770,148.580
C04391=1176.141,293.247,-69.932,-176.860,7.773,148.580
C04392=1176.137,293.495,-69.962,-176.858,7.775,148.580
C04393=1176.133,293.743,-69.992,-176.856,7.778,148.580
C04394=1176.129,293.992,-70.021,-176.853,7.781,148.580
C04395=1176.124,294.240,-70.052,-176.850,7.784,148.580
C04396=1176.120,294.488,-70.081,-176.848,7.788,148.580
C04397=1176.116,294.737,-70.111,-176.845,7.791,148.580
C04398=1176.112,294.984,-70.141,-176.842,7.794,148.580
C04399=1176.107,295.233,-70.171,-176.840,7.797,148.580
C04400=1176.103,295.481,-70.201,-176.837,7.799,148.580
C04401=1176.099,295.729,-70.231,-176.835,7.802,148.580
C04402=1176.095,295.977,-70.260,-176.832,7.805,148.580
C04403=1176.090,296.226,-70.290,-176.830,7.808,148.580
C04404=1176.086,296.473,-70.321,-176.827,7.811,148.580
C04405=1176.082,296.722,-70.350,-176.824,7.814,148.580
C04406=1176.078,296.970,-70.381,-176.822,7.817,148.580
C04407=1176.073,297.218,-70.410,-176.819,7.820,148.580
C04408=1176.069,297.466,-70.440,-176.817,7.823,148.580
C04409=1176.065,297.714,-70.471,-176.814,7.826,148.580
C04410=1176.060,297.962,-70.500,-176.812,7.829,148.580
C04411=1176.056,298.211,-70.531,-176.809,7.832,148.580
C04412=1176.052,298.459,-70.561,-176.807,7.835,148.580
C04413=1176.048,298.707,-70.591,-176.804,7.838,148.580
C04414=1176.044,298.955,-70.621,-176.802,7.841,148.580
C04415=1176.040,299.203,-70.651,-176.799,7.844,148.580
C04416=1176.035,299.451,-70.682,-176.796,7.847,148.580
C04417=1176.031,299.699,-70.711,-176.793,7.850,148.580
C04418=1176.026,299.947,-70.742,-176.791,7.853,148.580
C04419=1176.022,300.196,-70.771,-176.788,7.856,148.580
C04420=1176.018,300.444,-70.803,-176.786,7.858,148.580
C04421=1176.014,300.692,-70.833,-176.784,7.861,148.580
C04422=1176.010,300.940,-70.862,-176.781,7.865,148.580
C04423=1176.005,301.188,-70.893,-176.779,7.868,148.580
C04424=1176.001,301.436,-70.923,-176.776,7.871,148.580
C04425=1175.996,301.684,-70.953,-176.773,7.874,148.580
C04426=1175.993,301.933,-70.984,-176.771,7.877,148.581
C04427=1175.989,302.181,-71.014,-176.768,7.880,148.581
C04428=1175.984,302.429,-71.044,-176.765,7.883,148.581
C04429=1175.980,302.677,-71.075,-176.763,7.886,148.581
C04430=1175.975,302.925,-71.105,-176.760,7.889,148.581
C04431=1175.972,303.173,-71.136,-176.758,7.892,148.581
C04432=1175.967,303.422,-71.166,-176.755,7.895,148.581
C04433=1175.963,303.670,-71.196,-176.753,7.898,148.581
C04434=1175.958,303.917,-71.227,-176.750,7.901,148.581
C04435=1175.954,304.165,-71.258,-176.748,7.904,148.581
C04436=1175.951,304.414,-71.288,-176.745,7.907,148.581
C04437=1175.946,304.662,-71.319,-176.743,7.910,148.581
C04438=1175.942,304.910,-71.348,-176.740,7.913,148.581
C04439=1175.937,305.158,-71.379,-176.737,7.916,148.581
C04440=1175.933,305.407,-71.410,-176.735,7.919,148.581
C04441=1175.929,305.654,-71.440,-176.732,7.922,148.581
C04442=1175.925,305.902,-71.471,-176.730,7.925,148.581
C04443=1175.920,306.150,-71.502,-176.727,7.928,148.581
C04444=1175.917,306.399,-71.533,-176.725,7.931,148.581
C04445=1175.912,306.646,-71.563,-176.722,7.934,148.581
C04446=1175.908,306.894,-71.594,-176.720,7.938,148.581
C04447=1175.904,307.142,-71.624,-176.717,7.941,148.581
C04448=1175.900,307.391,-71.655,-176.714,7.944,148.581
C04449=1175.895,307.639,-71.686,-176.712,7.946,148.581
C04450=1175.890,307.887,-71.717,-176.710,7.949,148.581
C04451=1175.887,308.135,-71.747,-176.707,7.952,148.581
C04452=1175.883,308.383,-71.778,-176.705,7.955,148.582
C04453=1175.878,308.631,-71.809,-176.702,7.958,148.582
C04454=1175.873,308.879,-71.840,-176.699,7.961,148.582
C04455=1175.870,309.127,-71.870,-176.697,7.965,148.582
C04456=1175.865,309.375,-71.901,-176.694,7.968,148.582
C04457=1175.861,309.623,-71.932,-176.692,7.971,148.582
C04458=1175.857,309.872,-71.963,-176.689,7.974,148.582
C04459=1175.853,310.119,-71.993,-176.686,7.977,148.582
C04460=1175.848,310.367,-72.024,-176.684,7.980,148.582
C04461=1175.845,310.615,-72.056,-176.681,7.983,148.582
C04462=1175.840,310.863,-72.086,-176.679,7.986,148.582
C04463=1175.836,311.112,-72.118,-176.676,7.990,148.582
C04464=1175.831,311.360,-72.148,-176.674,7.993,148.582
C04465=1175.828,311.608,-72.179,-176.671,7.996,148.582
C04466=1175.824,311.856,-72.210,-176.669,7.999,148.582
C04467=1175.819,312.104,-72.241,-176.666,8.002,148.582
C04468=1175.815,312.352,-72.272,-176.664,8.005,148.583
C04469=1175.811,312.600,-72.303,-176.661,8.008,148.583
C04470=1175.806,312.848,-72.335,-176.658,8.011,148.583
C04471=1175.802,313.096,-72.366,-176.656,8.014,148.583
C04472=1175.798,313.344,-72.396,-176.653,8.017,148.583
C04473=1175.793,313.592,-72.428,-176.651,8.021,148.583
C04474=1175.789,313.869,-72.462,-176.648,8.024,148.583
C04475=1175.784,314.146,-72.497,-176.646,8.027,148.583
C04476=1175.780,314.422,-72.532,-176.643,8.031,148.583
C04477=1175.775,314.699,-72.566,-176.640,8.034,148.583
C04478=1175.771,314.948,-72.598,-176.638,8.037,148.583
C04479=1175.766,315.195,-72.629,-176.635,8.040,148.583
C04480=1175.763,315.444,-72.661,-176.632,8.043,148.583
C04481=1175.758,315.691,-72.691,-176.630,8.046,148.584
C04482=1175.754,315.940,-72.723,-176.627,8.049,148.584
C04483=1175.750,316.187,-72.754,-176.625,8.053,148.584
C04484=1175.746,316.436,-72.785,-176.622,8.056,148.584
C04485=1175.741,316.683,-72.817,-176.620,8.059,148.584
C04486=1175.737,316.932,-72.848,-176.617,8.062,148.584
C04487=1175.733,317.179,-72.879,-176.615,8.065,148.584
C04488=1175.729,317.428,-72.910,-176.612,8.068,148.584
C04489=1175.725,317.675,-72.942,-176.610,8.071,148.584
C04490=1175.721,317.923,-72.974,-176.607,8.075,148.584
C04491=1175.716,318.171,-73.004,-176.605,8.078,148.584
C04492=1175.713,318.419,-73.036,-176.602,8.081,148.584
C04493=1175.708,318.667,-73.067,-176.600,8.084,148.584
C04494=1175.704,318.915,-73.099,-176.597,8.087,148.585
C04495=1175.700,319.163,-73.130,-176.595,8.090,148.585
C04496=1175.696,319.411,-73.162,-176.592,8.093,148.585
C04497=1175.692,319.659,-73.193,-176.590,8.096,148.585
C04498=1175.688,319.907,-73.224,-176.587,8.100,148.585
C04499=1175.683,320.155,-73.256,-176.585,8.103,148.585
C04500=1175.679,320.403,-73.288,-176.582,8.106,148.585
C04501=1175.675,320.650,-73.320,-176.580,8.109,148.585
C04502=1175.671,320.899,-73.351,-176.577,8.112,148.585
C04503=1175.667,321.147,-73.383,-176.575,8.115,148.585
C04504=1175.663,321.395,-73.414,-176.572,8.119,148.586
C04505=1175.658,321.644,-73.446,-176.570,8.122,148.586
C04506=1175.653,321.891,-73.477,-176.567,8.125,148.586
C04507=1175.650,322.139,-73.509,-176.565,8.128,148.586
C04508=1175.646,322.387,-73.541,-176.562,8.131,148.586
C04509=1175.642,322.634,-73.572,-176.560,8.134,148.586
C04510=1175.637,322.883,-73.604,-176.557,8.138,148.586
C04511=1175.633,323.131,-73.636,-176.555,8.141,148.586
C04512=1175.629,323.379,-73.667,-176.552,8.144,148.586
C04513=1175.625,323.627,-73.699,-176.550,8.147,148.587
C04514=1175.621,323.874,-73.731,-176.547,8.151,148.587
C04515=1175.617,324.122,-73.763,-176.544,8.154,148.587
C04516=1175.613,324.370,-73.795,-176.542,8.157,148.587
C04517=1175.609,324.618,-73.827,-176.539,8.161,148.587
C04518=1175.604,324.866,-73.859,-176.537,8.164,148.587
C04519=1175.600,325.115,-73.890,-176.534,8.167,148.587
C04520=1175.596,325.362,-73.922,-176.532,8.170,148.587
C04521=1175.592,325.610,-73.953,-176.529,8.173,148.587
C04522=1175.588,325.858,-73.986,-176.527,8.176,148.588
C04523=1175.583,326.106,-74.017,-176.524,8.179,148.588
C04524=1175.580,326.354,-74.049,-176.522,8.183,148.588
C04525=1175.575,326.602,-74.082,-176.519,8.186,148.588
C04526=1175.571,326.850,-74.113,-176.517,8.189,148.588
C04527=1175.566,327.098,-74.146,-176.515,8.192,148.588
C04528=1175.563,327.345,-74.178,-176.512,8.195,148.588
C04529=1175.559,327.593,-74.210,-176.510,8.199,148.588
C04530=1175.554,327.841,-74.242,-176.507,8.202,148.588
C04531=1175.551,328.089,-74.274,-176.505,8.205,148.589
C04532=1175.546,328.337,-74.306,-176.503,8.208,148.589
C04533=1175.542,328.585,-74.338,-176.500,8.211,148.589
C04534=1175.538,328.833,-74.370,-176.498,8.215,148.589
C04535=1175.534,329.081,-74.402,-176.495,8.218,148.589
C04536=1175.530,329.329,-74.434,-176.493,8.221,148.589
C04537=1175.525,329.576,-74.467,-176.490,8.224,148.589
C04538=1175.521,329.824,-74.499,-176.488,8.227,148.590
C04539=1175.517,330.073,-74.531,-176.485,8.230,148.590
C04540=1175.513,330.321,-74.563,-176.483,8.235,148.590
C04541=1175.509,330.568,-74.596,-176.480,8.238,148.590
C04542=1175.505,330.816,-74.627,-176.478,8.241,148.590
C04543=1175.500,331.064,-74.660,-176.475,8.244,148.590
C04544=1175.497,331.312,-74.692,-176.473,8.247,148.590
C04545=1175.492,331.559,-74.725,-176.470,8.250,148.590
C04546=1175.488,331.807,-74.756,-176.468,8.254,148.591
C04547=1175.484,332.055,-74.789,-176.466,8.257,148.591
C04548=1175.480,332.303,-74.821,-176.463,8.260,148.591
C04549=1175.476,332.551,-74.854,-176.461,8.263,148.591
C04550=1175.471,332.799,-74.886,-176.458,8.267,148.591
C04551=1175.468,333.046,-74.918,-176.456,8.270,148.591
C04552=1175.463,333.295,-74.951,-176.453,8.273,148.592
C04553=1175.459,333.543,-74.983,-176.451,8.276,148.592
C04554=1175.455,333.790,-75.016,-176.449,8.280,148.592
C04555=1175.452,334.038,-75.048,-176.446,8.283,148.592
C04556=1175.447,334.285,-75.081,-176.443,8.287,148.592
C04557=1175.442,334.534,-75.113,-176.441,8.290,148.592
C04558=1175.439,334.781,-75.146,-176.438,8.293,148.592
C04559=1175.435,335.030,-75.178,-176.436,8.296,148.593
C04560=1175.430,335.278,-75.210,-176.434,8.300,148.593
C04561=1175.427,335.525,-75.243,-176.432,8.303,148.593
C04562=1175.423,335.773,-75.276,-176.429,8.306,148.593
C04563=1175.418,336.021,-75.308,-176.427,8.309,148.593
C04564=1175.414,336.268,-75.341,-176.424,8.313,148.593
C04565=1175.410,336.517,-75.373,-176.422,8.316,148.594
C04566=1175.406,336.764,-75.406,-176.420,8.319,148.594
C04567=1175.402,337.012,-75.438,-176.417,8.322,148.594
C04568=1175.398,337.260,-75.471,-176.414,8.326,148.594
C04569=1175.394,337.508,-75.505,-176.412,8.330,148.594
C04570=1175.389,337.756,-75.537,-176.410,8.333,148.595
C04571=1175.386,338.003,-75.570,-176.407,8.336,148.595
C04572=1175.381,338.252,-75.602,-176.405,8.339,148.595
C04573=1175.377,338.500,-75.635,-176.402,8.342,148.595
C04574=1175.372,338.747,-75.668,-176.400,8.346,148.595
C04575=1175.369,338.995,-75.700,-176.398,8.349,148.595
C04576=1175.365,339.242,-75.733,-176.396,8.352,148.596
C04577=1175.360,339.490,-75.766,-176.393,8.356,148.596
C04578=1175.356,339.770,-75.804,-176.390,8.360,148.596
C04579=1175.351,340.048,-75.840,-176.387,8.364,148.596
C04580=1175.346,340.328,-75.877,-176.385,8.367,148.596
C04581=1175.342,340.607,-75.914,-176.382,8.371,148.597
C04582=1175.338,340.855,-75.947,-176.380,8.374,148.597
C04583=1175.334,341.102,-75.980,-176.377,8.378,148.597
C04584=1175.330,341.350,-76.013,-176.375,8.381,148.597
C04585=1175.325,341.598,-76.046,-176.372,8.384,148.597
C04586=1175.321,341.846,-76.079,-176.370,8.387,148.597
C04587=1175.317,342.094,-76.112,-176.367,8.391,148.598
C04588=1175.313,342.342,-76.145,-176.365,8.395,148.598
C04589=1175.309,342.589,-76.177,-176.363,8.398,148.598
C04590=1175.305,342.837,-76.211,-176.361,8.401,148.598
C04591=1175.301,343.085,-76.244,-176.358,8.405,148.599
C04592=1175.297,343.332,-76.277,-176.356,8.408,148.599
C04593=1175.293,343.580,-76.310,-176.354,8.411,148.599
C04594=1175.289,343.828,-76.343,-176.351,8.415,148.599
C04595=1175.284,344.076,-76.376,-176.349,8.419,148.599
C04596=1175.280,344.323,-76.410,-176.346,8.422,148.600
C04597=1175.276,344.571,-76.443,-176.344,8.425,148.600
C04598=1175.273,344.819,-76.476,-176.342,8.429,148.600
C04599=1175.269,345.067,-76.509,-176.339,8.432,148.600
C04600=1175.264,345.315,-76.543,-176.337,8.435,148.601
C04601=1175.260,345.563,-76.576,-176.335,8.439,148.601
C04602=1175.256,345.810,-76.609,-176.333,8.442,148.601
C04603=1175.252,346.058,-76.642,-176.330,8.446,148.601
C04604=1175.248,346.306,-76.675,-176.328,8.449,148.601
C04605=1175.244,346.554,-76.708,-176.325,8.453,148.602
C04606=1175.240,346.801,-76.742,-176.323,8.456,148.602
C04607=1175.235,347.049,-76.775,-176.321,8.459,148.602
C04608=1175.231,347.297,-76.808,-176.318,8.463,148.602
C04609=1175.227,347.544,-76.841,-176.316,8.466,148.603
C04610=1175.224,347.792,-76.875,-176.313,8.470,148.603
C04611=1175.219,348.040,-76.909,-176.311,8.473,148.603
C04612=1175.215,348.288,-76.942,-176.309,8.477,148.603
C04613=1175.211,348.536,-76.975,-176.307,8.480,148.603
C04614=1175.207,348.783,-77.008,-176.304,8.483,148.604
C04615=1175.203,349.031,-77.042,-176.302,8.486,148.604
C04616=1175.199,349.278,-77.075,-176.300,8.490,148.604
C04617=1175.195,349.527,-77.109,-176.297,8.494,148.604
C04618=1175.191,349.774,-77.142,-176.295,8.497,148.605
C04619=1175.186,350.022,-77.177,-176.292,8.501,148.605
C04620=1175.182,350.270,-77.210,-176.290,8.504,148.605
C04621=1175.178,350.517,-77.243,-176.288,8.507,148.605
C04622=1175.174,350.764,-77.277,-176.286,8.511,148.606
C04623=1175.171,351.013,-77.310,-176.283,8.515,148.606
C04624=1175.167,351.261,-77.343,-176.281,8.518,148.606
C04625=1175.162,351.508,-77.378,-176.279,8.521,148.606
C04626=1175.158,351.756,-77.411,-176.276,8.525,148.607
C04627=1175.154,352.003,-77.444,-176.274,8.528,148.607
C04628=1175.151,352.251,-77.478,-176.272,8.532,148.607
C04629=1175.146,352.499,-77.512,-176.269,8.536,148.607
C04630=1175.142,352.746,-77.546,-176.267,8.539,148.608
C04631=1175.138,352.994,-77.579,-176.265,8.542,148.608
C04632=1175.134,353.241,-77.613,-176.263,8.546,148.608
C04633=1175.130,353.490,-77.647,-176.261,8.549,148.609
C04634=1175.126,353.737,-77.681,-176.258,8.553,148.609
C04635=1175.122,353.985,-77.714,-176.256,8.557,148.609
C04636=1175.118,354.232,-77.748,-176.254,8.560,148.609
C04637=1175.114,354.481,-77.782,-176.251,8.564,148.610
C04638=1175.110,354.728,-77.816,-176.249,8.567,148.610
C04639=1175.106,354.976,-77.849,-176.247,8.570,148.610
C04640=1175.101,355.223,-77.884,-176.244,8.575,148.611
C04641=1175.097,355.471,-77.917,-176.242,8.578,148.611
C04642=1175.094,355.719,-77.951,-176.240,8.581,148.611
C04643=1175.089,355.966,-77.986,-176.238,8.585,148.611
C04644=1175.086,356.214,-78.019,-176.236,8.588,148.612
C04645=1175.082,356.461,-78.053,-176.233,8.592,148.612
C04646=1175.077,356.709,-78.087,-176.231,8.596,148.612
C04647=1175.073,356.957,-78.121,-176.229,8.599,148.613
C04648=1175.069,357.205,-78.155,-176.227,8.603,148.613
C04649=1175.065,357.452,-78.189,-176.224,8.606,148.613
C04650=1175.061,357.700,-78.222,-176.222,8.610,148.614
C04651=1175.057,357.948,-78.257,-176.220,8.614,148.614
C04652=1175.053,358.195,-78.291,-176.218,8.617,148.614
C04653=1175.048,358.443,-78.325,-176.216,8.621,148.614
C04654=1175.045,358.691,-78.359,-176.213,8.624,148.615
C04655=1175.041,358.938,-78.394,-176.211,8.628,148.615
C04656=1175.037,359.185,-78.428,-176.209,8.632,148.615
C04657=1175.033,359.433,-78.462,-176.207,8.635,148.616
C04658=1175.029,359.681,-78.496,-176.204,8.639,148.616
C04659=1175.025,359.929,-78.530,-176.203,8.642,148.616
C04660=1175.021,360.176,-78.564,-176.200,8.646,148.617
C04661=1175.017,360.423,-78.598,-176.198,8.650,148.617
C04662=1175.013,360.672,-78.633,-176.196,8.653,148.617
C04663=1175.009,360.919,-78.667,-176.194,8.657,148.618
C04664=1175.005,361.166,-78.701,-176.192,8.660,148.618
C04665=1175.001,361.414,-78.735,-176.190,8.664,148.618
C04666=1174.997,361.662,-78.769,-176.187,8.668,148.619
C04667=1174.993,361.910,-78.803,-176.185,8.672,148.619
C04668=1174.989,362.157,-78.838,-176.183,8.675,148.620
C04669=1174.985,362.405,-78.873,-176.181,8.678,148.620
C04670=1174.981,362.652,-78.907,-176.179,8.682,148.620
C04671=1174.976,362.900,-78.941,-176.177,8.686,148.621
C04672=1174.973,363.148,-78.975,-176.175,8.689,148.621
C04673=1174.969,363.395,-79.010,-176.173,8.693,148.621
C04674=1174.965,363.643,-79.044,-176.171,8.697,148.622
C04675=1174.961,363.890,-79.079,-176.169,8.701,148.622
C04676=1174.957,364.138,-79.113,-176.167,8.704,148.622
C04677=1174.953,364.385,-79.147,-176.165,8.708,148.623
C04678=1174.949,364.634,-79.182,-176.163,8.711,148.623
C04679=1174.945,364.880,-79.217,-176.161,8.715,148.624
C04680=1174.941,365.128,-79.251,-176.159,8.718,148.624
C04681=1174.937,365.376,-79.286,-176.157,8.722,148.624
C04682=1174.932,365.657,-79.325,-176.155,8.726,148.625
C04683=1174.928,365.940,-79.364,-176.152,8.731,148.625
C04684=1174.923,366.222,-79.403,-176.151,8.735,148.626
C04685=1174.918,366.503,-79.443,-176.148,8.739,148.626
C04686=1174.914,366.751,-79.478,-176.147,8.743,148.627
C04687=1174.911,366.998,-79.512,-176.145,8.746,148.627
C04688=1174.907,367.246,-79.547,-176.143,8.750,148.628
C04689=1174.902,367.493,-79.582,-176.141,8.753,148.628
C04690=1174.899,367.741,-79.616,-176.139,8.757,148.629
C04691=1174.895,367.988,-79.651,-176.137,8.761,148.629
C04692=1174.891,368.236,-79.686,-176.136,8.764,148.629
C04693=1174.886,368.483,-79.720,-176.134,8.768,148.630
C04694=1174.883,368.731,-79.754,-176.132,8.771,148.630
C04695=1174.879,368.979,-79.790,-176.130,8.775,148.631
C04696=1174.875,369.226,-79.825,-176.129,8.779,148.631
C04697=1174.871,369.474,-79.859,-176.127,8.783,148.632
C04698=1174.867,369.721,-79.895,-176.125,8.786,148.632
C04699=1174.863,369.969,-79.929,-176.123,8.790,148.633
C04700=1174.859,370.216,-79.963,-176.122,8.794,148.633
C04701=1174.855,370.464,-79.999,-176.120,8.797,148.634
C04702=1174.851,370.711,-80.033,-176.118,8.801,148.634
C04703=1174.847,370.959,-80.068,-176.116,8.805,148.635
C04704=1174.843,371.207,-80.104,-176.115,8.808,148.635
C04705=1174.839,371.454,-80.137,-176.114,8.811,148.636
C04706=1174.835,371.701,-80.173,-176.112,8.815,148.636
C04707=1174.831,371.949,-80.207,-176.110,8.819,148.637
C04708=1174.827,372.197,-80.242,-176.109,8.823,148.637
C04709=1174.823,372.445,-80.278,-176.107,8.826,148.638
C04710=1174.819,372.692,-80.312,-176.105,8.830,148.638
C04711=1174.815,372.939,-80.348,-176.104,8.833,148.639
C04712=1174.811,373.187,-80.382,-176.103,8.837,148.639
C04713=1174.808,373.434,-80.417,-176.101,8.841,148.640
C04714=1174.804,373.682,-80.452,-176.100,8.844,148.640
C04715=1174.799,373.929,-80.487,-176.099,8.847,148.641
C04716=1174.795,374.177,-80.522,-176.097,8.851,148.641
C04717=1174.791,374.424,-80.557,-176.096,8.855,148.642
C04718=1174.787,374.671,-80.593,-176.094,8.859,148.642
C04719=1174.783,374.920,-80.628,-176.093,8.862,148.643
C04720=1174.779,375.166,-80.663,-176.092,8.866,148.644
C04721=1174.775,375.414,-80.698,-176.090,8.869,148.644
C04722=1174.772,375.662,-80.733,-176.089,8.872,148.645
C04723=1174.767,375.909,-80.768,-176.088,8.876,148.645
C04724=1174.763,376.157,-80.803,-176.087,8.879,148.646
C04725=1174.760,376.404,-80.839,-176.085,8.883,148.647
C04726=1174.755,376.652,-80.873,-176.083,8.887,148.647
C04727=1174.751,376.899,-80.909,-176.083,8.890,148.648
C04728=1174.748,377.147,-80.944,-176.081,8.894,148.648
C04729=1174.743,377.394,-80.979,-176.080,8.897,148.649
C04730=1174.740,377.642,-81.014,-176.079,8.901,148.649
C04731=1174.736,377.889,-81.050,-176.078,8.904,148.650
C04732=1174.731,378.137,-81.084,-176.077,8.908,148.651
C04733=1174.728,378.384,-81.120,-176.076,8.911,148.651
C04734=1174.724,378.632,-81.156,-176.075,8.915,148.652
C04735=1174.720,378.878,-81.191,-176.074,8.918,148.652
C04736=1174.716,379.127,-81.226,-176.072,8.922,148.653
C04737=1174.712,379.374,-81.261,-176.071,8.925,148.654
C04738=1174.708,379.622,-81.297,-176.070,8.929,148.654
C04739=1174.704,379.868,-81.332,-176.069,8.932,148.655
C04740=1174.700,380.116,-81.367,-176.068,8.935,148.655
C04741=1174.697,380.364,-81.402,-176.067,8.939,148.656
C04742=1174.692,380.611,-81.437,-176.067,8.942,148.657
C04743=1174.689,380.858,-81.473,-176.066,8.946,148.657
C04744=1174.685,381.106,-81.508,-176.065,8.949,148.658
C04745=1174.680,381.354,-81.544,-176.064,8.953,148.659
C04746=1174.676,381.601,-81.579,-176.063,8.956,148.659
C04747=1174.672,381.849,-81.615,-176.062,8.959,148.660
C04748=1174.669,382.096,-81.650,-176.061,8.962,148.660
C04749=1174.665,382.344,-81.686,-176.060,8.966,148.661
C04750=1174.661,382.590,-81.721,-176.060,8.969,148.662
C04751=1174.657,382.838,-81.756,-176.059,8.973,148.662
C04752=1174.653,383.086,-81.791,-176.058,8.976,148.663
C04753=1174.649,383.334,-81.827,-176.058,8.979,148.664
C04754=1174.644,383.581,-81.863,-176.057,8.982,148.664
C04755=1174.641,383.828,-81.898,-176.056,8.985,148.665
C04756=1174.637,384.076,-81.934,-176.056,8.989,148.666
C04757=1174.633,384.323,-81.969,-176.055,8.992,148.666
C04758=1174.629,384.570,-82.004,-176.054,8.995,148.667
C04759=1174.625,384.818,-82.041,-176.053,8.998,148.668
C04760=1174.621,385.065,-82.076,-176.053,9.002,148.668
C04761=1174.617,385.313,-82.112,-176.052,9.005,148.669
C04762=1174.614,385.560,-82.147,-176.052,9.008,148.670
C04763=1174.610,385.807,-82.182,-176.051,9.011,148.670
C04764=1174.606,386.054,-82.218,-176.051,9.015,148.671
C04765=1174.601,386.302,-82.254,-176.050,9.018,148.672
C04766=1174.598,386.550,-82.289,-176.049,9.021,148.673
C04767=1174.594,386.798,-82.324,-176.049,9.024,148.673
C04768=1174.590,387.044,-82.360,-176.049,9.027,148.674
C04769=1174.586,387.292,-82.396,-176.048,9.030,148.675
C04770=1174.582,387.539,-82.432,-176.047,9.033,148.675
C04771=1174.578,387.787,-82.468,-176.048,9.036,148.676
C04772=1174.574,388.034,-82.503,-176.047,9.039,148.677
C04773=1174.570,388.281,-82.538,-176.046,9.042,148.677
C04774=1174.566,388.529,-82.574,-176.046,9.045,148.678
C04775=1174.562,388.776,-82.610,-176.046,9.048,148.679
C04776=1174.559,389.024,-82.646,-176.046,9.052,148.680
C04777=1174.555,389.271,-82.681,-176.045,9.054,148.680
C04778=1174.550,389.519,-82.717,-176.045,9.057,148.681
C04779=1174.546,389.766,-82.752,-176.045,9.060,148.682
C04780=1174.543,390.014,-82.788,-176.044,9.063,148.682
C04781=1174.539,390.261,-82.824,-176.044,9.065,148.683
C04782=1174.534,390.509,-82.860,-176.044,9.069,148.684
C04783=1174.531,390.756,-82.895,-176.044,9.071,148.684
C04784=1174.527,391.003,-82.931,-176.044,9.075,148.685
C04785=1174.523,391.250,-82.967,-176.044,9.077,148.686
C04786=1174.518,391.535,-83.008,-176.044,9.081,148.687
C04787=1174.514,391.820,-83.049,-176.043,9.084,148.687
C04788=1174.510,392.104,-83.090,-176.043,9.087,148.688
C04789=1174.505,392.389,-83.132,-176.043,9.090,148.689
C04790=1174.501,392.636,-83.167,-176.043,9.093,148.690
C04791=1174.497,392.884,-83.203,-176.043,9.096,148.690
C04792=1174.493,393.131,-83.239,-176.043,9.099,148.691
C04793=1174.489,393.378,-83.274,-176.043,9.101,148.692
C04794=1174.485,393.626,-83.310,-176.043,9.103,148.692
C04795=1174.481,393.873,-83.346,-176.042,9.107,148.693
C04796=1174.478,394.120,-83.382,-176.042,9.109,148.694
C04797=1174.474,394.368,-83.418,-176.043,9.112,148.695
C04798=1174.470,394.616,-83.454,-176.043,9.115,148.695
C04799=1174.466,394.863,-83.489,-176.043,9.117,148.696
C04800=1174.462,395.110,-83.524,-176.043,9.119,148.696
C04801=1174.458,395.357,-83.561,-176.043,9.122,148.697
C04802=1174.454,395.605,-83.597,-176.042,9.125,148.698
C04803=1174.450,395.852,-83.632,-176.043,9.128,148.699
C04804=1174.446,396.100,-83.669,-176.043,9.130,148.699
C04805=1174.442,396.348,-83.704,-176.042,9.133,148.700
C04806=1174.439,396.594,-83.740,-176.043,9.135,148.701
C04807=1174.434,396.842,-83.776,-176.043,9.138,148.701
C04808=1174.430,397.089,-83.812,-176.043,9.140,148.702
C04809=1174.426,397.337,-83.848,-176.043,9.143,148.703
C04810=1174.422,397.584,-83.884,-176.043,9.146,148.703
C04811=1174.419,397.831,-83.920,-176.043,9.148,148.704
C04812=1174.414,398.079,-83.956,-176.043,9.150,148.705
C04813=1174.411,398.327,-83.991,-176.043,9.153,148.705
C04814=1174.407,398.573,-84.028,-176.044,9.155,148.706
C04815=1174.403,398.821,-84.064,-176.044,9.157,148.707
C04816=1174.399,399.068,-84.099,-176.044,9.160,148.707
C04817=1174.394,399.316,-84.135,-176.044,9.162,148.708
C04818=1174.391,399.563,-84.171,-176.044,9.165,148.709
C04819=1174.387,399.810,-84.207,-176.044,9.167,148.709
C04820=1174.383,400.058,-84.243,-176.045,9.170,148.710
C04821=1174.379,400.305,-84.279,-176.045,9.171,148.711
C04822=1174.376,400.552,-84.315,-176.045,9.174,148.711
C04823=1174.371,400.800,-84.351,-176.045,9.176,148.712
C04824=1174.368,401.048,-84.386,-176.045,9.179,148.713
C04825=1174.364,401.295,-84.423,-176.045,9.181,148.713
C04826=1174.359,401.542,-84.459,-176.046,9.183,148.714
C04827=1174.356,401.789,-84.494,-176.046,9.186,148.715
C04828=1174.352,402.036,-84.531,-176.046,9.188,148.715
C04829=1174.348,402.284,-84.566,-176.046,9.190,148.716
C04830=1174.344,402.532,-84.603,-176.047,9.192,148.717
C04831=1174.340,402.779,-84.639,-176.047,9.195,148.717
C04832=1174.337,403.026,-84.674,-176.046,9.197,148.718
C04833=1174.332,403.274,-84.711,-176.047,9.199,148.718
C04834=1174.329,403.521,-84.747,-176.047,9.201,148.719
C04835=1174.324,403.769,-84.783,-176.047,9.204,148.720
C04836=1174.321,404.016,-84.819,-176.048,9.205,148.720
C04837=1174.317,404.263,-84.855,-176.048,9.208,148.721
C04838=1174.312,404.510,-84.891,-176.048,9.210,148.722
C04839=1174.309,404.758,-84.926,-176.048,9.212,148.722
C04840=1174.305,405.005,-84.963,-176.048,9.214,148.723
C04841=1174.301,405.252,-84.999,-176.049,9.216,148.724
C04842=1174.297,405.500,-85.035,-176.049,9.218,148.724
C04843=1174.293,405.747,-85.071,-176.049,9.221,148.725
C04844=1174.289,405.995,-85.107,-176.049,9.222,148.725
C04845=1174.285,406.242,-85.143,-176.050,9.225,148.726
C04846=1174.282,406.489,-85.179,-176.050,9.227,148.727
C04847=1174.277,406.737,-85.215,-176.050,9.229,148.727
C04848=1174.274,406.984,-85.251,-176.051,9.231,148.728
C04849=1174.270,407.232,-85.287,-176.050,9.233,148.728
C04850=1174.266,407.479,-85.323,-176.051,9.235,148.729
C04851=1174.262,407.726,-85.360,-176.051,9.237,148.730
C04852=1174.258,407.973,-85.395,-176.052,9.239,148.730
C04853=1174.254,408.220,-85.431,-176.052,9.241,148.731
C04854=1174.250,408.468,-85.467,-176.052,9.243,148.731
C04855=1174.246,408.715,-85.503,-176.052,9.245,148.732
C04856=1174.242,408.963,-85.540,-176.052,9.247,148.733
C04857=1174.238,409.210,-85.575,-176.053,9.249,148.733
C04858=1174.234,409.457,-85.612,-176.053,9.251,148.734
C04859=1174.231,409.705,-85.648,-176.053,9.253,148.734
C04860=1174.226,409.953,-85.684,-176.053,9.255,148.735
C04861=1174.223,410.199,-85.720,-176.054,9.257,148.736
C04862=1174.219,410.447,-85.756,-176.054,9.259,148.736
C04863=1174.215,410.694,-85.793,-176.054,9.261,148.737
C04864=1174.211,410.942,-85.829,-176.054,9.263,148.737
C04865=1174.207,411.189,-85.864,-176.055,9.264,148.738
C04866=1174.203,411.437,-85.901,-176.055,9.267,148.738
C04867=1174.199,411.684,-85.937,-176.055,9.268,148.739
C04868=1174.196,411.931,-85.973,-176.055,9.271,148.740
C04869=1174.192,412.179,-86.009,-176.055,9.272,148.740
C04870=1174.188,412.426,-86.045,-176.055,9.274,148.741
C04871=1174.183,412.673,-86.081,-176.056,9.276,148.741
C04872=1174.180,412.920,-86.117,-176.056,9.278,148.742
C04873=1174.175,413.167,-86.154,-176.056,9.280,148.742
C04874=1174.172,413.415,-86.189,-176.057,9.282,148.743
C04875=1174.168,413.662,-86.226,-176.057,9.283,148.743
C04876=1174.164,413.910,-86.262,-176.057,9.286,148.744
C04877=1174.160,414.157,-86.298,-176.057,9.287,148.744
C04878=1174.156,414.404,-86.334,-176.057,9.289,148.745
C04879=1174.152,414.652,-86.371,-176.058,9.291,148.746
C04880=1174.149,414.899,-86.406,-176.058,9.293,148.746
C04881=1174.144,415.146,-86.443,-176.058,9.295,148.747
C04882=1174.141,415.394,-86.479,-176.058,9.297,148.747
C04883=1174.137,415.641,-86.516,-176.059,9.298,148.748
C04884=1174.134,415.889,-86.551,-176.058,9.300,148.748
C04885=1174.133,416.135,-86.588,-176.059,9.302,148.749
C04886=1174.132,416.392,-86.624,-176.059,9.303,148.749
C04887=1174.134,416.649,-86.661,-176.059,9.305,148.750
C04888=1174.135,416.905,-86.698,-176.059,9.307,148.750
C04889=1174.138,417.160,-86.735,-176.060,9.309,148.751
C04890=1173.717,417.162,-86.779,-176.063,9.319,148.754
C04891=1173.714,416.903,-86.742,-176.062,9.318,148.754
C04892=1173.712,416.644,-86.705,-176.062,9.316,148.753
C04893=1173.712,416.384,-86.667,-176.062,9.314,148.753
C04894=1173.712,416.125,-86.629,-176.062,9.313,148.752
C04895=1173.713,415.877,-86.593,-176.062,9.311,148.752
C04896=1173.716,415.630,-86.557,-176.062,9.309,148.751
C04897=1173.720,415.382,-86.521,-176.061,9.307,148.751
C04898=1173.723,415.135,-86.485,-176.061,9.306,148.750
C04899=1173.727,414.888,-86.449,-176.061,9.303,148.750
C04900=1173.731,414.641,-86.413,-176.061,9.302,148.749
C04901=1173.735,414.393,-86.376,-176.060,9.300,148.749
C04902=1173.738,414.146,-86.340,-176.060,9.298,148.748
C04903=1173.743,413.898,-86.304,-176.060,9.296,148.748
C04904=1173.746,413.651,-86.268,-176.060,9.295,148.747
C04905=1173.751,413.403,-86.232,-176.059,9.292,148.746
C04906=1173.755,413.157,-86.196,-176.059,9.291,148.746
C04907=1173.759,412.909,-86.160,-176.059,9.289,148.745
C04908=1173.763,412.662,-86.124,-176.059,9.287,148.745
C04909=1173.767,412.415,-86.087,-176.058,9.285,148.744
C04910=1173.770,412.167,-86.052,-176.058,9.283,148.744
C04911=1173.774,411.920,-86.015,-176.058,9.281,148.743
C04912=1173.778,411.673,-85.979,-176.058,9.279,148.743
C04913=1173.782,411.425,-85.942,-176.058,9.277,148.742
C04914=1173.786,411.178,-85.907,-176.057,9.276,148.742
C04915=1173.790,410.931,-85.870,-176.057,9.273,148.741
C04916=1173.794,410.683,-85.834,-176.057,9.272,148.740
C04917=1173.798,410.435,-85.798,-176.057,9.269,148.740
C04918=1173.801,410.189,-85.762,-176.056,9.268,148.739
C04919=1173.806,409.941,-85.726,-176.056,9.265,148.738
C04920=1173.809,409.694,-85.690,-176.056,9.264,148.738
C04921=1173.814,409.446,-85.653,-176.055,9.262,148.737
C04922=1173.817,409.199,-85.617,-176.056,9.260,148.737
C04923=1173.821,408.951,-85.581,-176.055,9.258,148.736
C04924=1173.825,408.704,-85.545,-176.055,9.256,148.736
C04925=1173.828,408.457,-85.509,-176.054,9.254,148.735
C04926=1173.833,408.209,-85.473,-176.055,9.252,148.734
C04927=1173.837,407.963,-85.437,-176.054,9.250,148.734
C04928=1173.841,407.715,-85.401,-176.054,9.248,148.733
C04929=1173.845,407.468,-85.365,-176.053,9.246,148.733
C04930=1173.849,407.220,-85.329,-176.053,9.244,148.732
C04931=1173.852,406.973,-85.293,-176.053,9.242,148.731
C04932=1173.857,406.726,-85.256,-176.053,9.240,148.731
C04933=1173.860,406.478,-85.221,-176.053,9.238,148.730
C04934=1173.865,406.230,-85.184,-176.052,9.236,148.730
C04935=1173.868,405.984,-85.148,-176.052,9.234,148.729
C04936=1173.872,405.736,-85.113,-176.052,9.232,148.728
C04937=1173.876,405.488,-85.077,-176.052,9.229,148.728
C04938=1173.879,405.241,-85.040,-176.052,9.228,148.727
C04939=1173.884,404.994,-85.004,-176.051,9.225,148.727
C04940=1173.887,404.747,-84.968,-176.051,9.223,148.726
C04941=1173.892,404.499,-84.932,-176.051,9.221,148.725
C04942=1173.895,404.251,-84.896,-176.051,9.218,148.725
C04943=1173.899,404.005,-84.860,-176.050,9.217,148.724
C04944=1173.904,403.757,-84.824,-176.050,9.214,148.723
C04945=1173.907,403.510,-84.789,-176.050,9.213,148.723
C04946=1173.911,403.263,-84.752,-176.049,9.210,148.722
C04947=1173.915,403.015,-84.716,-176.049,9.208,148.721
C04948=1173.919,402.767,-84.680,-176.049,9.206,148.721
C04949=1173.923,402.521,-84.644,-176.049,9.204,148.720
C04950=1173.926,402.273,-84.608,-176.049,9.201,148.720
C04951=1173.931,402.025,-84.572,-176.049,9.198,148.719
C04952=1173.934,401.778,-84.536,-176.048,9.197,148.718
C04953=1173.939,401.531,-84.500,-176.048,9.194,148.718
C04954=1173.942,401.283,-84.464,-176.048,9.192,148.717
C04955=1173.946,401.037,-84.428,-176.048,9.189,148.716
C04956=1173.951,400.789,-84.392,-176.048,9.188,148.716
C04957=1173.954,400.542,-84.357,-176.047,9.185,148.715
C04958=1173.958,400.294,-84.320,-176.047,9.183,148.714
C04959=1173.962,400.047,-84.284,-176.047,9.180,148.714
C04960=1173.966,399.799,-84.249,-176.047,9.178,148.713
C04961=1173.970,399.552,-84.212,-176.047,9.176,148.712
C04962=1173.973,399.305,-84.176,-176.046,9.174,148.712
C04963=1173.978,399.057,-84.140,-176.046,9.171,148.711
C04964=1173.982,398.809,-84.104,-176.046,9.168,148.710
C04965=1173.985,398.563,-84.069,-176.046,9.166,148.710
C04966=1173.990,398.315,-84.032,-176.046,9.164,148.709
C04967=1173.994,398.068,-83.997,-176.046,9.161,148.708
C04968=1173.997,397.820,-83.961,-176.046,9.159,148.708
C04969=1174.001,397.573,-83.924,-176.046,9.156,148.707
C04970=1174.005,397.326,-83.889,-176.045,9.154,148.706
C04971=1174.009,397.078,-83.853,-176.045,9.152,148.706
C04972=1174.013,396.830,-83.817,-176.045,9.149,148.705
C04973=1174.016,396.583,-83.781,-176.045,9.147,148.704
C04974=1174.021,396.336,-83.745,-176.045,9.144,148.704
C04975=1174.025,396.089,-83.710,-176.045,9.142,148.703
C04976=1174.029,395.841,-83.674,-176.045,9.138,148.702
C04977=1174.033,395.594,-83.637,-176.045,9.136,148.701
C04978=1174.036,395.347,-83.602,-176.045,9.133,148.701
C04979=1174.040,395.099,-83.566,-176.045,9.131,148.700
C04980=1174.045,394.851,-83.530,-176.045,9.128,148.699
C04981=1174.048,394.604,-83.494,-176.045,9.126,148.699
C04982=1174.052,394.358,-83.459,-176.045,9.123,148.698
C04983=1174.057,394.110,-83.422,-176.044,9.121,148.697
C04984=1174.060,393.862,-83.387,-176.045,9.117,148.696
C04985=1174.064,393.615,-83.351,-176.045,9.115,148.696
C04986=1174.068,393.367,-83.315,-176.045,9.112,148.695
C04987=1174.072,393.120,-83.279,-176.045,9.110,148.695
C04988=1174.075,392.873,-83.243,-176.045,9.106,148.694
C04989=1174.080,392.626,-83.208,-176.045,9.104,148.693
C04990=1174.084,392.378,-83.172,-176.045,9.101,148.692
C04991=1174.089,392.093,-83.131,-176.045,9.098,148.692
C04992=1174.093,391.809,-83.090,-176.045,9.095,148.691
C04993=1174.097,391.524,-83.049,-176.046,9.092,148.690
C04994=1174.102,391.239,-83.007,-176.046,9.088,148.689
C04995=1174.106,390.992,-82.972,-176.046,9.086,148.689
C04996=1174.109,390.744,-82.936,-176.046,9.083,148.688
C04997=1174.113,390.497,-82.900,-176.046,9.080,148.687
C04998=1174.118,390.250,-82.865,-176.046,9.077,148.686
C04999=1174.121,390.003,-82.828,-176.046,9.074,148.686
C05000=1174.125,389.756,-82.793,-176.047,9.071,148.685
C05001=1174.129,389.508,-82.757,-176.047,9.068,148.684
C05002=1174.133,389.260,-82.721,-176.047,9.065,148.684
C05003=1174.137,389.013,-82.686,-176.047,9.062,148.683
C05004=1174.141,388.766,-82.650,-176.048,9.059,148.682
C05005=1174.145,388.518,-82.615,-176.048,9.056,148.681
C05006=1174.149,388.271,-82.579,-176.048,9.053,148.681
C05007=1174.153,388.023,-82.543,-176.049,9.050,148.680
C05008=1174.156,387.776,-82.508,-176.050,9.047,148.679
C05009=1174.160,387.528,-82.472,-176.049,9.044,148.679
C05010=1174.165,387.281,-82.436,-176.050,9.041,148.678
C05011=1174.169,387.033,-82.401,-176.051,9.038,148.677
C05012=1174.172,386.786,-82.365,-176.051,9.034,148.677
C05013=1174.176,386.538,-82.330,-176.051,9.032,148.676
C05014=1174.180,386.291,-82.294,-176.052,9.029,148.675
C05015=1174.185,386.044,-82.258,-176.052,9.025,148.674
C05016=1174.188,385.796,-82.223,-176.053,9.022,148.674
C05017=1174.192,385.549,-82.187,-176.053,9.019,148.673
C05018=1174.196,385.301,-82.152,-176.054,9.016,148.673
C05019=1174.199,385.054,-82.116,-176.055,9.012,148.672
C05020=1174.204,384.807,-82.080,-176.055,9.009,148.671
C05021=1174.208,384.559,-82.045,-176.056,9.006,148.670
C05022=1174.212,384.312,-82.009,-176.057,9.003,148.670
C05023=1174.215,384.064,-81.974,-176.057,8.999,148.669
C05024=1174.220,383.817,-81.939,-176.058,8.996,148.668
C05025=1174.224,383.570,-81.902,-176.058,8.993,148.668
C05026=1174.228,383.322,-81.867,-176.059,8.990,148.667
C05027=1174.231,383.075,-81.831,-176.060,8.987,148.667
C05028=1174.235,382.827,-81.796,-176.060,8.983,148.666
C05029=1174.239,382.580,-81.761,-176.061,8.980,148.665
C05030=1174.243,382.332,-81.726,-176.062,8.977,148.665
C05031=1174.247,382.085,-81.690,-176.063,8.973,148.664
C05032=1174.251,381.837,-81.654,-176.064,8.970,148.663
C05033=1174.256,381.590,-81.619,-176.065,8.967,148.663
C05034=1174.259,381.343,-81.583,-176.066,8.964,148.662
C05035=1174.263,381.095,-81.548,-176.067,8.960,148.661
C05036=1174.268,380.848,-81.513,-176.067,8.956,148.661
C05037=1174.271,380.600,-81.478,-176.068,8.953,148.660
C05038=1174.275,380.353,-81.442,-176.070,8.949,148.659
C05039=1174.278,380.105,-81.407,-176.070,8.946,148.659
C05040=1174.283,379.858,-81.372,-176.071,8.943,148.658
C05041=1174.287,379.610,-81.337,-176.072,8.939,148.657
C05042=1174.290,379.363,-81.301,-176.073,8.936,148.657
C05043=1174.295,379.115,-81.265,-176.074,8.933,148.656
C05044=1174.299,378.868,-81.230,-176.075,8.929,148.656
C05045=1174.303,378.621,-81.194,-176.076,8.926,148.655
C05046=1174.307,378.373,-81.159,-176.078,8.922,148.654
C05047=1174.311,378.126,-81.124,-176.078,8.919,148.654
C05048=1174.315,377.878,-81.089,-176.080,8.915,148.653
C05049=1174.319,377.630,-81.054,-176.081,8.912,148.653
C05050=1174.323,377.383,-81.019,-176.082,8.908,148.652
C05051=1174.327,377.136,-80.983,-176.083,8.905,148.651
C05052=1174.330,376.888,-80.948,-176.084,8.901,148.651
C05053=1174.335,376.641,-80.913,-176.086,8.897,148.650
C05054=1174.338,376.393,-80.878,-176.087,8.894,148.650
C05055=1174.342,376.145,-80.843,-176.088,8.890,148.649
C05056=1174.347,375.898,-80.808,-176.089,8.887,148.649
C05057=1174.350,375.651,-80.772,-176.091,8.883,148.648
C05058=1174.354,375.403,-80.737,-176.092,8.880,148.648
C05059=1174.359,375.156,-80.702,-176.093,8.877,148.647
C05060=1174.362,374.908,-80.667,-176.095,8.873,148.646
C05061=1174.366,374.660,-80.632,-176.096,8.869,148.646
C05062=1174.370,374.414,-80.596,-176.097,8.866,148.645
C05063=1174.374,374.166,-80.562,-176.099,8.862,148.645
C05064=1174.377,373.918,-80.527,-176.100,8.858,148.644
C05065=1174.382,373.671,-80.492,-176.102,8.855,148.644
C05066=1174.386,373.423,-80.457,-176.103,8.851,148.643
C05067=1174.390,373.176,-80.422,-176.105,8.848,148.643
C05068=1174.394,372.928,-80.387,-176.106,8.844,148.642
C05069=1174.398,372.680,-80.352,-176.108,8.840,148.642
C05070=1174.402,372.434,-80.317,-176.109,8.836,148.641
C05071=1174.406,372.185,-80.282,-176.111,8.833,148.640
C05072=1174.410,371.938,-80.246,-176.112,8.830,148.640
C05073=1174.413,371.691,-80.212,-176.114,8.826,148.639
C05074=1174.417,371.443,-80.177,-176.115,8.822,148.639
C05075=1174.422,371.196,-80.142,-176.117,8.819,148.638
C05076=1174.426,370.948,-80.108,-176.119,8.815,148.638
C05077=1174.430,370.701,-80.072,-176.120,8.811,148.637
C05078=1174.434,370.453,-80.038,-176.122,8.807,148.637
C05079=1174.437,370.206,-80.003,-176.124,8.804,148.637
C05080=1174.441,369.958,-79.968,-176.125,8.800,148.636
C05081=1174.445,369.710,-79.933,-176.127,8.796,148.635
C05082=1174.450,369.463,-79.898,-176.128,8.794,148.635
C05083=1174.454,369.215,-79.863,-176.130,8.790,148.635
C05084=1174.457,368.968,-79.829,-176.132,8.786,148.634
C05085=1174.461,368.721,-79.794,-176.134,8.782,148.634
C05086=1174.466,368.473,-79.759,-176.135,8.779,148.633
C05087=1174.470,368.225,-79.725,-176.137,8.775,148.633
C05088=1174.474,367.977,-79.690,-176.139,8.772,148.632
C05089=1174.477,367.730,-79.655,-176.141,8.768,148.632
C05090=1174.481,367.482,-79.620,-176.143,8.764,148.631
C05091=1174.486,367.235,-79.586,-176.145,8.760,148.631
C05092=1174.490,366.987,-79.551,-176.147,8.756,148.631
C05093=1174.493,366.740,-79.516,-176.149,8.753,148.630
C05094=1174.497,366.492,-79.482,-176.151,8.749,148.630
C05095=1174.502,366.211,-79.442,-176.152,8.745,148.629
C05096=1174.507,365.929,-79.403,-176.155,8.741,148.629
C05097=1174.511,365.646,-79.364,-176.157,8.737,148.628
C05098=1174.516,365.365,-79.325,-176.159,8.733,148.628
C05099=1174.520,365.116,-79.290,-176.161,8.729,148.627
C05100=1174.523,364.869,-79.256,-176.163,8.725,148.627
C05101=1174.527,364.622,-79.220,-176.165,8.721,148.627
C05102=1174.532,364.374,-79.186,-176.167,8.718,148.626
C05103=1174.535,364.127,-79.152,-176.169,8.714,148.626
C05104=1174.539,363.879,-79.117,-176.171,8.711,148.625
C05105=1174.543,363.632,-79.083,-176.173,8.707,148.625
C05106=1174.547,363.384,-79.049,-176.175,8.704,148.625
C05107=1174.552,363.137,-79.014,-176.177,8.700,148.624
C05108=1174.555,362.889,-78.980,-176.180,8.696,148.624
C05109=1174.560,362.641,-78.945,-176.181,8.692,148.623
C05110=1174.563,362.394,-78.911,-176.184,8.689,148.623
C05111=1174.567,362.146,-78.877,-176.185,8.685,148.623
C05112=1174.572,361.899,-78.842,-176.187,8.682,148.622
C05113=1174.575,361.651,-78.808,-176.190,8.678,148.622
C05114=1174.580,361.403,-78.774,-176.192,8.674,148.622
C05115=1174.583,361.156,-78.739,-176.194,8.671,148.621
C05116=1174.588,360.908,-78.705,-176.196,8.667,148.621
C05117=1174.592,360.661,-78.672,-176.198,8.664,148.621
C05118=1174.596,360.412,-78.637,-176.200,8.660,148.620
C05119=1174.600,360.165,-78.603,-176.203,8.656,148.620
C05120=1174.604,359.917,-78.568,-176.205,8.652,148.620
C05121=1174.607,359.670,-78.534,-176.207,8.649,148.619
C05122=1174.612,359.423,-78.500,-176.209,8.645,148.619
C05123=1174.615,359.174,-78.466,-176.211,8.642,148.619
C05124=1174.620,358.927,-78.432,-176.214,8.638,148.618
C05125=1174.624,358.680,-78.398,-176.216,8.634,148.618
C05126=1174.627,358.432,-78.364,-176.218,8.631,148.618
C05127=1174.632,358.184,-78.329,-176.220,8.627,148.617
C05128=1174.636,357.937,-78.296,-176.222,8.624,148.617
C05129=1174.640,357.689,-78.261,-176.225,8.620,148.617
C05130=1174.644,357.442,-78.227,-176.227,8.616,148.617
C05131=1174.648,357.193,-78.194,-176.229,8.613,148.616
C05132=1174.652,356.946,-78.159,-176.231,8.609,148.616
C05133=1174.656,356.699,-78.126,-176.233,8.606,148.616
C05134=1174.660,356.451,-78.091,-176.236,8.602,148.615
C05135=1174.664,356.203,-78.058,-176.238,8.598,148.615
C05136=1174.667,355.956,-78.024,-176.240,8.595,148.615
C05137=1174.672,355.708,-77.990,-176.243,8.592,148.615
C05138=1174.676,355.460,-77.956,-176.244,8.588,148.614
C05139=1174.679,355.213,-77.922,-176.247,8.584,148.614
C05140=1174.684,354.965,-77.888,-176.250,8.581,148.614
C05141=1174.688,354.717,-77.854,-176.251,8.577,148.613
C05142=1174.692,354.469,-77.821,-176.254,8.574,148.613
C05143=1174.696,354.222,-77.786,-176.256,8.571,148.613
C05144=1174.700,353.974,-77.753,-176.259,8.566,148.612
C05145=1174.704,353.727,-77.719,-176.261,8.563,148.612
C05146=1174.708,353.478,-77.685,-176.263,8.560,148.612
C05147=1174.712,353.231,-77.651,-176.265,8.556,148.612
C05148=1174.716,352.983,-77.618,-176.267,8.553,148.611
C05149=1174.720,352.736,-77.584,-176.270,8.549,148.611
C05150=1174.725,352.487,-77.550,-176.272,8.545,148.611
C05151=1174.728,352.240,-77.516,-176.274,8.542,148.610
C05152=1174.733,351.993,-77.483,-176.277,8.539,148.610
C05153=1174.736,351.745,-77.449,-176.279,8.535,148.610
C05154=1174.741,351.497,-77.415,-176.281,8.532,148.610
C05155=1174.745,351.249,-77.382,-176.284,8.528,148.610
C05156=1174.749,351.002,-77.348,-176.286,8.524,148.609
C05157=1174.753,350.754,-77.315,-176.288,8.521,148.609
C05158=1174.757,350.506,-77.282,-176.290,8.518,148.609
C05159=1174.761,350.259,-77.247,-176.293,8.514,148.608
C05160=1174.765,350.011,-77.214,-176.295,8.511,148.608
C05161=1174.769,349.763,-77.181,-176.298,8.507,148.608
C05162=1174.773,349.516,-77.147,-176.300,8.504,148.608
C05163=1174.777,349.268,-77.113,-176.302,8.500,148.608
C05164=1174.781,349.020,-77.080,-176.305,8.497,148.607
C05165=1174.785,348.773,-77.047,-176.307,8.493,148.607
C05166=1174.790,348.525,-77.013,-176.309,8.490,148.607
C05167=1174.793,348.277,-76.979,-176.312,8.486,148.606
C05168=1174.798,348.029,-76.946,-176.314,8.483,148.606
C05169=1174.802,347.781,-76.913,-176.316,8.479,148.606
C05170=1174.806,347.533,-76.880,-176.318,8.476,148.606
C05171=1174.810,347.286,-76.847,-176.321,8.473,148.606
C05172=1174.814,347.039,-76.813,-176.323,8.469,148.605
C05173=1174.818,346.791,-76.780,-176.325,8.466,148.605
C05174=1174.822,346.543,-76.746,-176.328,8.462,148.605
C05175=1174.826,346.295,-76.713,-176.330,8.459,148.605
C05176=1174.830,346.047,-76.680,-176.333,8.455,148.604
C05177=1174.834,345.799,-76.647,-176.335,8.452,148.604
C05178=1174.838,345.552,-76.613,-176.337,8.449,148.604
C05179=1174.842,345.304,-76.580,-176.340,8.445,148.604
C05180=1174.846,345.056,-76.547,-176.342,8.442,148.604
C05181=1174.850,344.808,-76.514,-176.345,8.438,148.603
C05182=1174.855,344.561,-76.481,-176.347,8.435,148.603
C05183=1174.859,344.313,-76.448,-176.349,8.431,148.603
C05184=1174.863,344.065,-76.414,-176.351,8.428,148.603
C05185=1174.867,343.817,-76.381,-176.354,8.425,148.602
C05186=1174.871,343.570,-76.348,-176.356,8.421,148.602
C05187=1174.875,343.322,-76.315,-176.358,8.418,148.602
C05188=1174.879,343.074,-76.282,-176.361,8.414,148.602
C05189=1174.884,342.827,-76.249,-176.363,8.411,148.602
C05190=1174.888,342.579,-76.216,-176.366,8.408,148.602
C05191=1174.892,342.331,-76.182,-176.368,8.404,148.601
C05192=1174.896,342.083,-76.149,-176.371,8.401,148.601
C05193=1174.900,341.836,-76.116,-176.373,8.398,148.601
C05194=1174.905,341.587,-76.084,-176.375,8.394,148.601
C05195=1174.909,341.340,-76.050,-176.377,8.391,148.600
C05196=1174.912,341.092,-76.018,-176.380,8.388,148.600
C05197=1174.916,340.844,-75.985,-176.383,8.384,148.600
C05198=1174.920,340.597,-75.952,-176.385,8.380,148.600
C05199=1174.925,340.317,-75.914,-176.387,8.377,148.600
C05200=1174.930,340.038,-75.878,-176.390,8.373,148.600
C05201=1174.934,339.758,-75.841,-176.393,8.369,148.599
C05202=1174.940,339.479,-75.804,-176.396,8.366,148.599
C05203=1174.943,339.232,-75.771,-176.398,8.363,148.599
C05204=1174.947,338.984,-75.738,-176.400,8.359,148.599
C05205=1174.952,338.736,-75.705,-176.403,8.355,148.598
C05206=1174.956,338.488,-75.672,-176.406,8.352,148.598
C05207=1174.960,338.240,-75.639,-176.408,8.349,148.598
C05208=1174.964,337.992,-75.607,-176.410,8.346,148.598
C05209=1174.968,337.745,-75.574,-176.413,8.342,148.598
C05210=1174.972,337.497,-75.541,-176.415,8.339,148.598
C05211=1174.976,337.249,-75.509,-176.418,8.336,148.598
C05212=1174.980,337.001,-75.476,-176.420,8.333,148.597
C05213=1174.985,336.754,-75.444,-176.422,8.329,148.597
C05214=1174.989,336.506,-75.411,-176.424,8.326,148.597
C05215=1174.992,336.258,-75.378,-176.427,8.322,148.597
C05216=1174.997,336.010,-75.346,-176.430,8.319,148.597
C05217=1175.001,335.762,-75.313,-176.432,8.316,148.596
C05218=1175.005,335.514,-75.281,-176.434,8.312,148.596
C05219=1175.009,335.267,-75.248,-176.437,8.309,148.596
C05220=1175.013,335.018,-75.215,-176.439,8.306,148.596
C05221=1175.017,334.772,-75.183,-176.442,8.303,148.596
C05222=1175.022,334.523,-75.150,-176.444,8.299,148.596
C05223=1175.026,334.275,-75.117,-176.446,8.296,148.595
C05224=1175.029,334.027,-75.085,-176.449,8.293,148.595
C05225=1175.034,333.780,-75.052,-176.451,8.290,148.595
C05226=1175.037,333.532,-75.020,-176.454,8.286,148.595
C05227=1175.042,333.283,-74.988,-176.456,8.282,148.595
C05228=1175.046,333.036,-74.955,-176.459,8.279,148.595
C05229=1175.050,332.788,-74.923,-176.461,8.276,148.595
C05230=1175.055,332.540,-74.891,-176.464,8.273,148.594
C05231=1175.058,332.292,-74.858,-176.466,8.270,148.594
C05232=1175.062,332.044,-74.826,-176.469,8.266,148.594
C05233=1175.067,331.797,-74.794,-176.471,8.263,148.594
C05234=1175.071,331.549,-74.761,-176.474,8.260,148.594
C05235=1175.075,331.301,-74.729,-176.476,8.257,148.594
C05236=1175.079,331.053,-74.697,-176.478,8.254,148.594
C05237=1175.083,330.805,-74.664,-176.480,8.250,148.593
C05238=1175.087,330.558,-74.632,-176.483,8.247,148.593
C05239=1175.092,330.309,-74.600,-176.485,8.244,148.593
C05240=1175.096,330.061,-74.568,-176.488,8.241,148.593
C05241=1175.099,329.814,-74.536,-176.490,8.238,148.593
C05242=1175.104,329.566,-74.503,-176.493,8.234,148.593
C05243=1175.108,329.318,-74.472,-176.496,8.231,148.593
C05244=1175.112,329.070,-74.439,-176.498,8.227,148.592
C05245=1175.116,328.822,-74.407,-176.501,8.224,148.592
C05246=1175.121,328.574,-74.375,-176.503,8.221,148.592
C05247=1175.124,328.327,-74.343,-176.506,8.218,148.592
C05248=1175.129,328.078,-74.310,-176.508,8.214,148.592
C05249=1175.132,327.830,-74.278,-176.511,8.211,148.592
C05250=1175.137,327.583,-74.247,-176.513,8.208,148.592
C05251=1175.141,327.335,-74.214,-176.515,8.205,148.591
C05252=1175.145,327.086,-74.183,-176.518,8.202,148.591
C05253=1175.150,326.839,-74.151,-176.520,8.198,148.591
C05254=1175.154,326.591,-74.119,-176.523,8.195,148.591
C05255=1175.157,326.343,-74.087,-176.525,8.192,148.591
C05256=1175.162,326.095,-74.055,-176.527,8.189,148.591
C05257=1175.166,325.847,-74.023,-176.530,8.186,148.591
C05258=1175.170,325.599,-73.991,-176.532,8.183,148.591
C05259=1175.175,325.351,-73.959,-176.535,8.180,148.591
C05260=1175.179,325.103,-73.927,-176.537,8.176,148.590
C05261=1175.182,324.855,-73.895,-176.540,8.173,148.590
C05262=1175.187,324.608,-73.863,-176.542,8.170,148.590
C05263=1175.191,324.360,-73.831,-176.545,8.167,148.590
C05264=1175.195,324.112,-73.800,-176.547,8.164,148.590
C05265=1175.199,323.864,-73.768,-176.550,8.159,148.590
C05266=1175.204,323.616,-73.736,-176.553,8.157,148.590
C05267=1175.208,323.367,-73.705,-176.555,8.153,148.590
C05268=1175.212,323.120,-73.673,-176.558,8.150,148.590
C05269=1175.216,322.872,-73.641,-176.560,8.147,148.589
C05270=1175.220,322.624,-73.609,-176.563,8.144,148.589
C05271=1175.224,322.376,-73.577,-176.565,8.141,148.589
C05272=1175.228,322.128,-73.545,-176.568,8.138,148.589
C05273=1175.233,321.880,-73.515,-176.570,8.134,148.589
C05274=1175.236,321.632,-73.483,-176.572,8.131,148.589
C05275=1175.241,321.384,-73.450,-176.575,8.128,148.589
C05276=1175.245,321.136,-73.419,-176.577,8.125,148.589
C05277=1175.249,320.888,-73.388,-176.580,8.122,148.589
C05278=1175.253,320.640,-73.356,-176.582,8.118,148.588
C05279=1175.257,320.392,-73.324,-176.585,8.115,148.588
C05280=1175.261,320.145,-73.293,-176.587,8.112,148.588
C05281=1175.265,319.896,-73.262,-176.590,8.109,148.588
C05282=1175.270,319.648,-73.229,-176.592,8.106,148.588
C05283=1175.274,319.401,-73.198,-176.595,8.103,148.588
C05284=1175.278,319.152,-73.167,-176.597,8.100,148.588
C05285=1175.283,318.905,-73.135,-176.600,8.097,148.588
C05286=1175.287,318.656,-73.104,-176.602,8.093,148.588
C05287=1175.291,318.409,-73.073,-176.605,8.090,148.588
C05288=1175.295,318.161,-73.041,-176.607,8.087,148.587
C05289=1175.299,317.913,-73.010,-176.610,8.084,148.588
C05290=1175.303,317.665,-72.978,-176.613,8.081,148.588
C05291=1175.307,317.417,-72.947,-176.615,8.078,148.587
C05292=1175.311,317.169,-72.916,-176.618,8.075,148.587
C05293=1175.316,316.921,-72.885,-176.620,8.071,148.587
C05294=1175.319,316.673,-72.853,-176.623,8.068,148.587
C05295=1175.324,316.425,-72.822,-176.625,8.065,148.587
C05296=1175.328,316.177,-72.790,-176.628,8.062,148.587
C05297=1175.332,315.929,-72.760,-176.630,8.059,148.587
C05298=1175.336,315.681,-72.728,-176.633,8.056,148.587
C05299=1175.341,315.433,-72.697,-176.635,8.053,148.587
C05300=1175.344,315.185,-72.665,-176.638,8.050,148.587
C05301=1175.349,314.937,-72.634,-176.641,8.047,148.587
C05302=1175.353,314.688,-72.603,-176.643,8.043,148.586
C05303=1175.358,314.411,-72.568,-176.646,8.040,148.586
C05304=1175.362,314.135,-72.533,-176.649,8.036,148.586
C05305=1175.367,313.858,-72.498,-176.651,8.033,148.586
C05306=1175.373,313.581,-72.464,-176.655,8.029,148.586
C05307=1175.376,313.334,-72.433,-176.657,8.026,148.586
C05308=1175.380,313.086,-72.402,-176.660,8.023,148.586
C05309=1175.385,312.837,-72.371,-176.662,8.020,148.586
C05310=1175.389,312.590,-72.339,-176.665,8.017,148.586
C05311=1175.393,312.341,-72.308,-176.667,8.014,148.586
C05312=1175.397,312.093,-72.277,-176.670,8.010,148.586
C05313=1175.402,311.845,-72.247,-176.672,8.008,148.586
C05314=1175.406,311.597,-72.215,-176.674,8.005,148.586
C05315=1175.410,311.349,-72.184,-176.677,8.002,148.586
C05316=1175.414,311.101,-72.154,-176.679,7.999,148.586
C05317=1175.418,310.853,-72.123,-176.682,7.996,148.585
C05318=1175.423,310.605,-72.092,-176.684,7.993,148.585
C05319=1175.427,310.357,-72.060,-176.687,7.990,148.585
C05320=1175.431,310.109,-72.029,-176.689,7.986,148.585
C05321=1175.435,309.861,-71.999,-176.692,7.983,148.585
C05322=1175.439,309.612,-71.968,-176.694,7.980,148.585
C05323=1175.444,309.364,-71.937,-176.697,7.977,148.585
C05324=1175.448,309.117,-71.907,-176.700,7.974,148.585
C05325=1175.452,308.868,-71.875,-176.702,7.971,148.585
C05326=1175.456,308.620,-71.845,-176.705,7.968,148.585
C05327=1175.461,308.372,-71.815,-176.708,7.965,148.585
C05328=1175.465,308.124,-71.784,-176.710,7.962,148.585
C05329=1175.469,307.876,-71.753,-176.713,7.959,148.585
C05330=1175.473,307.628,-71.722,-176.715,7.956,148.585
C05331=1175.478,307.380,-71.692,-176.718,7.952,148.585
C05332=1175.482,307.131,-71.661,-176.720,7.949,148.585
C05333=1175.486,306.884,-71.630,-176.723,7.946,148.585
C05334=1175.490,306.636,-71.600,-176.725,7.943,148.584
C05335=1175.495,306.388,-71.569,-176.728,7.940,148.584
C05336=1175.499,306.139,-71.538,-176.731,7.937,148.584
C05337=1175.503,305.891,-71.508,-176.733,7.934,148.584
C05338=1175.508,305.644,-71.477,-176.735,7.932,148.584
C05339=1175.511,305.395,-71.446,-176.738,7.929,148.584
C05340=1175.515,305.147,-71.416,-176.740,7.925,148.584
C05341=1175.520,304.899,-71.385,-176.743,7.922,148.584
C05342=1175.524,304.652,-71.355,-176.746,7.919,148.584
C05343=1175.529,304.403,-71.325,-176.748,7.916,148.584
C05344=1175.533,304.154,-71.293,-176.751,7.913,148.584
C05345=1175.537,303.907,-71.263,-176.753,7.910,148.584
C05346=1175.541,303.659,-71.232,-176.756,7.907,148.584
C05347=1175.545,303.411,-71.202,-176.758,7.904,148.584
C05348=1175.549,303.162,-71.171,-176.761,7.901,148.584
C05349=1175.554,302.914,-71.141,-176.764,7.898,148.584
C05350=1175.558,302.666,-71.111,-176.766,7.894,148.584
C05351=1175.563,302.418,-71.080,-176.769,7.892,148.584
C05352=1175.567,302.170,-71.051,-176.772,7.889,148.584
C05353=1175.571,301.922,-71.020,-176.773,7.886,148.584
C05354=1175.575,301.674,-70.989,-176.776,7.883,148.584
C05355=1175.579,301.426,-70.959,-176.779,7.880,148.584
C05356=1175.583,301.177,-70.929,-176.782,7.877,148.584
C05357=1175.588,300.930,-70.898,-176.784,7.874,148.584
C05358=1175.592,300.682,-70.868,-176.787,7.871,148.584
C05359=1175.597,300.433,-70.838,-176.789,7.868,148.584
C05360=1175.600,300.185,-70.808,-176.792,7.865,148.584
C05361=1175.605,299.936,-70.778,-176.794,7.862,148.583
C05362=1175.609,299.689,-70.748,-176.797,7.859,148.583
C05363=1175.614,299.441,-70.717,-176.800,7.856,148.583
C05364=1175.618,299.193,-70.687,-176.802,7.853,148.583
C05365=1175.622,298.945,-70.657,-176.804,7.850,148.583
C05366=1175.627,298.696,-70.627,-176.807,7.847,148.583
C05367=1175.630,298.449,-70.597,-176.810,7.844,148.583
C05368=1175.635,298.199,-70.566,-176.812,7.841,148.583
C05369=1175.639,297.952,-70.536,-176.815,7.838,148.583
C05370=1175.643,297.703,-70.507,-176.817,7.835,148.583
C05371=1175.647,297.455,-70.476,-176.820,7.832,148.583
C05372=1175.652,297.207,-70.447,-176.823,7.829,148.583
C05373=1175.656,296.959,-70.416,-176.825,7.826,148.583
C05374=1175.660,296.711,-70.386,-176.828,7.823,148.583
C05375=1175.664,296.463,-70.356,-176.831,7.820,148.583
C05376=1175.669,296.215,-70.326,-176.833,7.817,148.583
C05377=1175.673,295.966,-70.297,-176.835,7.814,148.583
C05378=1175.677,295.719,-70.267,-176.838,7.811,148.583
C05379=1175.681,295.471,-70.237,-176.841,7.808,148.583
C05380=1175.685,295.222,-70.206,-176.843,7.805,148.583
C05381=1175.690,294.974,-70.177,-176.846,7.802,148.583
C05382=1175.694,294.725,-70.147,-176.848,7.799,148.583
C05383=1175.698,294.477,-70.116,-176.851,7.796,148.583
C05384=1175.703,294.229,-70.087,-176.854,7.793,148.583
C05385=1175.707,293.981,-70.057,-176.856,7.791,148.583
C05386=1175.711,293.733,-70.028,-176.859,7.788,148.583
C05387=1175.716,293.485,-69.997,-176.861,7.785,148.583
C05388=1175.720,293.236,-69.968,-176.864,7.782,148.583
C05389=1175.724,292.988,-69.938,-176.866,7.779,148.583
C05390=1175.728,292.740,-69.909,-176.869,7.776,148.583
C05391=1175.732,292.492,-69.879,-176.872,7.773,148.583
C05392=1175.737,292.244,-69.849,-176.875,7.770,148.583
C05393=1175.741,291.995,-69.819,-176.876,7.767,148.583
C05394=1175.745,291.747,-69.790,-176.879,7.764,148.583
C05395=1175.749,291.499,-69.760,-176.882,7.761,148.583
C05396=1175.753,291.251,-69.730,-176.884,7.758,148.583
C05397=1175.758,291.003,-69.701,-176.887,7.755,148.583
C05398=1175.762,290.754,-69.671,-176.890,7.752,148.583
C05399=1175.767,290.506,-69.641,-176.892,7.749,148.583
C05400=1175.771,290.259,-69.612,-176.895,7.746,148.583
C05401=1175.776,290.010,-69.583,-176.897,7.744,148.583
C05402=1175.780,289.762,-69.553,-176.900,7.741,148.583
C05403=1175.784,289.514,-69.524,-176.903,7.738,148.583
C05404=1175.788,289.265,-69.494,-176.905,7.735,148.583
C05405=1175.792,289.017,-69.465,-176.908,7.732,148.583
C05406=1175.796,288.769,-69.435,-176.910,7.729,148.583
C05407=1175.801,288.494,-69.402,-176.913,7.726,148.583
C05408=1175.807,288.219,-69.370,-176.916,7.723,148.583
C05409=1175.811,287.945,-69.337,-176.919,7.719,148.583
C05410=1175.816,287.670,-69.304,-176.922,7.716,148.583
C05411=1175.820,287.421,-69.275,-176.925,7.713,148.583
C05412=1175.824,287.174,-69.246,-176.927,7.711,148.583
C05413=1175.829,286.926,-69.216,-176.929,7.708,148.583
C05414=1175.833,286.677,-69.187,-176.932,7.705,148.583
C05415=1175.837,286.429,-69.158,-176.934,7.701,148.583
C05416=1175.841,286.181,-69.128,-176.937,7.698,148.583
C05417=1175.846,285.932,-69.099,-176.940,7.695,148.583
C05418=1175.850,285.684,-69.070,-176.943,7.692,148.583
C05419=1175.855,285.436,-69.041,-176.945,7.690,148.583
C05420=1175.859,285.188,-69.011,-176.948,7.687,148.583
C05421=1175.863,284.939,-68.982,-176.950,7.684,148.583
C05422=1175.867,284.691,-68.952,-176.953,7.681,148.583
C05423=1175.872,284.442,-68.924,-176.956,7.678,148.583
C05424=1175.876,284.194,-68.894,-176.958,7.675,148.583
C05425=1175.881,283.946,-68.865,-176.960,7.673,148.583
C05426=1175.885,283.698,-68.836,-176.963,7.670,148.583
C05427=1175.889,283.449,-68.807,-176.966,7.667,148.583
C05428=1175.893,283.201,-68.778,-176.968,7.664,148.583
C05429=1175.897,282.953,-68.749,-176.971,7.661,148.583
C05430=1175.902,282.706,-68.720,-176.974,7.658,148.583
C05431=1175.906,282.457,-68.691,-176.976,7.656,148.584
C05432=1175.910,282.208,-68.661,-176.979,7.653,148.584
C05433=1175.915,281.960,-68.632,-176.982,7.650,148.584
C05434=1175.920,281.712,-68.604,-176.984,7.647,148.584
C05435=1175.924,281.464,-68.574,-176.987,7.644,148.584
C05436=1175.928,281.215,-68.546,-176.989,7.642,148.584
C05437=1175.932,280.967,-68.517,-176.991,7.639,148.584
C05438=1175.937,280.719,-68.487,-176.994,7.636,148.584
C05439=1175.941,280.470,-68.459,-176.997,7.633,148.584
C05440=1175.945,280.222,-68.429,-177.000,7.630,148.584
C05441=1175.949,279.974,-68.401,-177.002,7.627,148.584
C05442=1175.954,279.726,-68.372,-177.005,7.624,148.584
C05443=1175.958,279.477,-68.343,-177.007,7.621,148.584
C05444=1175.962,279.229,-68.314,-177.010,7.619,148.584
C05445=1175.966,278.980,-68.286,-177.013,7.616,148.584
C05446=1175.971,278.733,-68.257,-177.015,7.613,148.584
C05447=1175.975,278.484,-68.228,-177.018,7.610,148.584
C05448=1175.980,278.236,-68.198,-177.020,7.607,148.584
C05449=1175.984,277.988,-68.171,-177.023,7.604,148.584
C05450=1175.988,277.739,-68.141,-177.026,7.601,148.584
C05451=1175.993,277.490,-68.112,-177.029,7.598,148.584
C05452=1175.996,277.243,-68.084,-177.031,7.596,148.584
C05453=1176.001,276.994,-68.055,-177.034,7.593,148.584
C05454=1176.006,276.745,-68.026,-177.036,7.590,148.584
C05455=1176.009,276.497,-67.998,-177.039,7.587,148.584
C05456=1176.014,276.249,-67.969,-177.041,7.585,148.585
C05457=1176.018,276.001,-67.940,-177.044,7.582,148.585
C05458=1176.023,275.753,-67.912,-177.047,7.579,148.585
C05459=1176.027,275.504,-67.883,-177.049,7.576,148.585
C05460=1176.031,275.256,-67.854,-177.052,7.573,148.585
C05461=1176.036,275.008,-67.826,-177.054,7.571,148.585
C05462=1176.040,274.759,-67.797,-177.057,7.568,148.585
C05463=1176.044,274.511,-67.769,-177.060,7.565,148.585
C05464=1176.049,274.263,-67.740,-177.062,7.562,148.585
C05465=1176.053,274.015,-67.712,-177.065,7.560,148.585
C05466=1176.058,273.766,-67.684,-177.067,7.557,148.585
C05467=1176.062,273.517,-67.655,-177.070,7.554,148.585
C05468=1176.066,273.269,-67.626,-177.073,7.551,148.585
C05469=1176.071,273.021,-67.598,-177.076,7.548,148.585
C05470=1176.074,272.773,-67.569,-177.078,7.546,148.585
C05471=1176.079,272.525,-67.541,-177.081,7.543,148.585
C05472=1176.083,272.276,-67.513,-177.083,7.540,148.585
C05473=1176.088,272.027,-67.484,-177.086,7.537,148.585
C05474=1176.092,271.780,-67.456,-177.088,7.535,148.586
C05475=1176.096,271.531,-67.427,-177.091,7.532,148.586
C05476=1176.101,271.283,-67.399,-177.094,7.529,148.586
